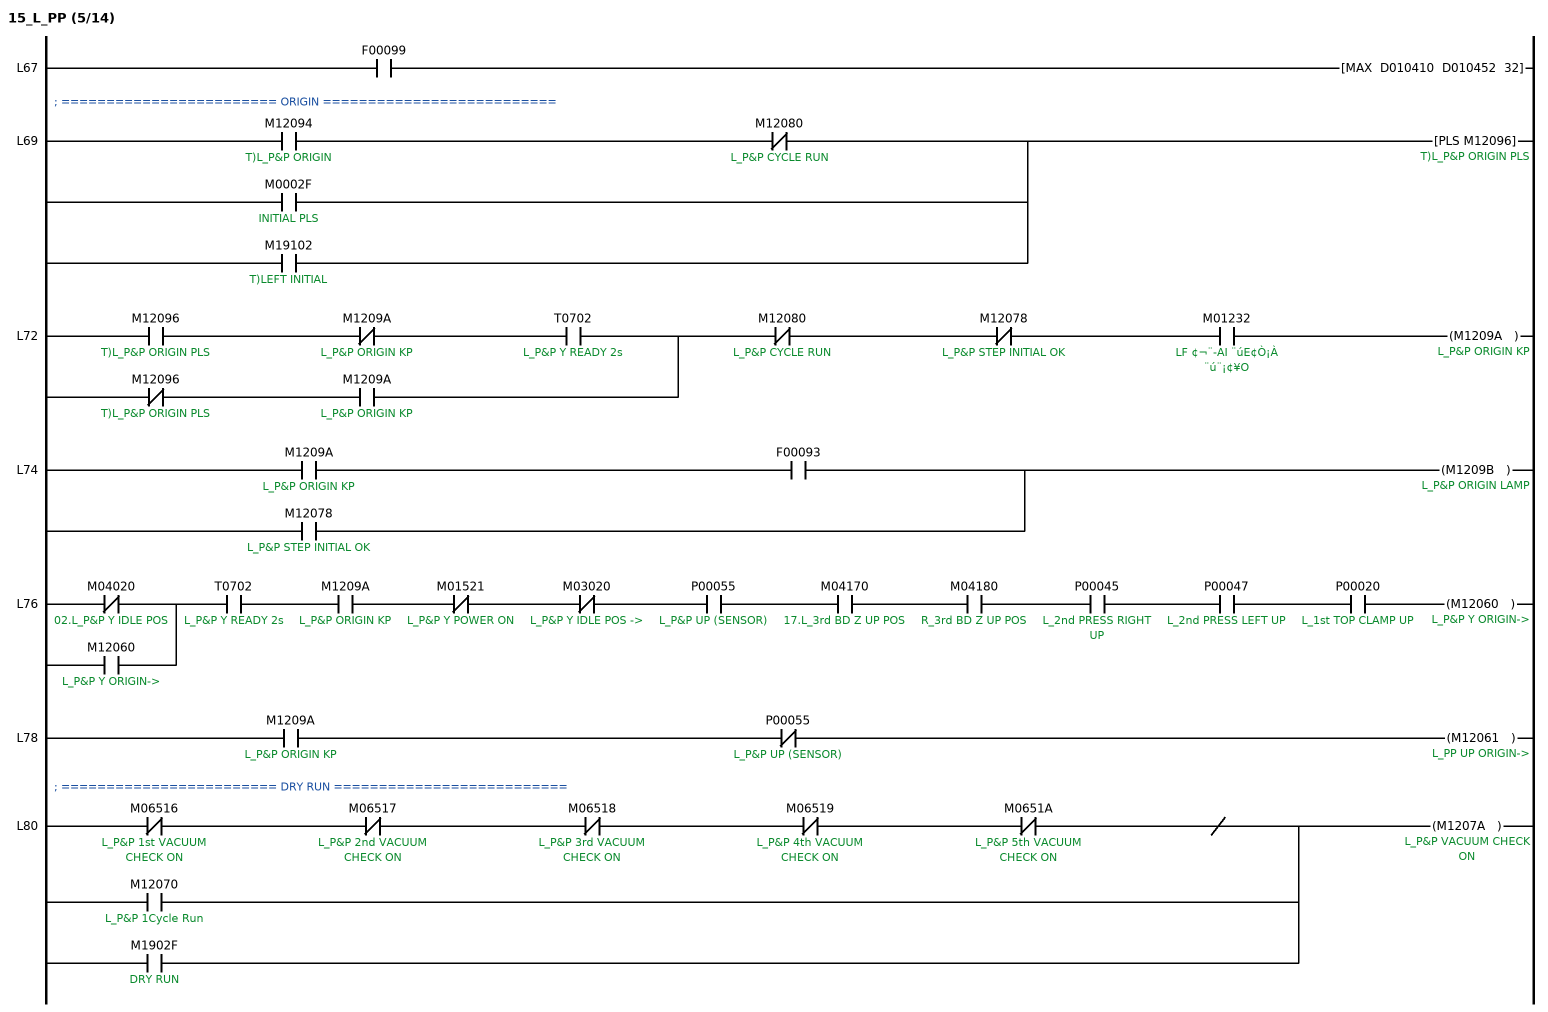
[picture p120: 15_L_PP rungs L67-L80]
; L67
LOAD      F00099
MAX       D010410 D010452 32
// ======================== ORIGIN ==========================
; L69
LOAD      M12094	// T)L_P&P ORIGIN
AND NOT   M12080	// L_P&P CYCLE RUN
OR        M0002F	// INITIAL PLS
OR        M19102	// T)LEFT INITIAL
OUTP      M12096	// T)L_P&P ORIGIN PLS
; L72
LOAD      M12096	// T)L_P&P ORIGIN PLS
AND NOT   M1209A	// L_P&P ORIGIN KP
AND       T0702	// L_P&P Y READY 2s
LOAD NOT  M12096	// T)L_P&P ORIGIN PLS
AND       M1209A	// L_P&P ORIGIN KP
OR LOAD
AND NOT   M12080	// L_P&P CYCLE RUN
AND NOT   M12078	// L_P&P STEP INITIAL OK
AND       M01232	// LF ¢¬¨­AI ¨úE¢Ò¡À ¨ú¨¡¢¥O
OUT       M1209A	// L_P&P ORIGIN KP
; L74
LOAD      M1209A	// L_P&P ORIGIN KP
AND       F00093
OR        M12078	// L_P&P STEP INITIAL OK
OUT       M1209B	// L_P&P ORIGIN LAMP
; L76
LOAD NOT  M04020	// 02.L_P&P Y IDLE POS
OR        M12060	// L_P&P Y ORIGIN->
AND       T0702	// L_P&P Y READY 2s
AND       M1209A	// L_P&P ORIGIN KP
AND NOT   M01521	// L_P&P Y POWER ON
AND NOT   M03020	// L_P&P Y IDLE POS ->
AND       P00055	// L_P&P UP (SENSOR)
AND       M04170	// 17.L_3rd BD Z UP POS
AND       M04180	// R_3rd BD Z UP POS
AND       P00045	// L_2nd PRESS RIGHT UP
AND       P00047	// L_2nd PRESS LEFT UP
AND       P00020	// L_1st TOP CLAMP UP
OUT       M12060	// L_P&P Y ORIGIN->
; L78
LOAD      M1209A	// L_P&P ORIGIN KP
AND NOT   P00055	// L_P&P UP (SENSOR)
OUT       M12061	// L_PP UP ORIGIN->
// ======================== DRY RUN ==========================
; L80
LOAD NOT  M06516	// L_P&P 1st VACUUM CHECK ON
AND NOT   M06517	// L_P&P 2nd VACUUM CHECK ON
AND NOT   M06518	// L_P&P 3rd VACUUM CHECK ON
AND NOT   M06519	// L_P&P 4th VACUUM CHECK ON
AND NOT   M0651A	// L_P&P 5th VACUUM CHECK ON
NOT
OR        M12070	// L_P&P 1Cycle Run
OR        M1902F	// DRY RUN
OUT       M1207A	// L_P&P VACUUM CHECK ON

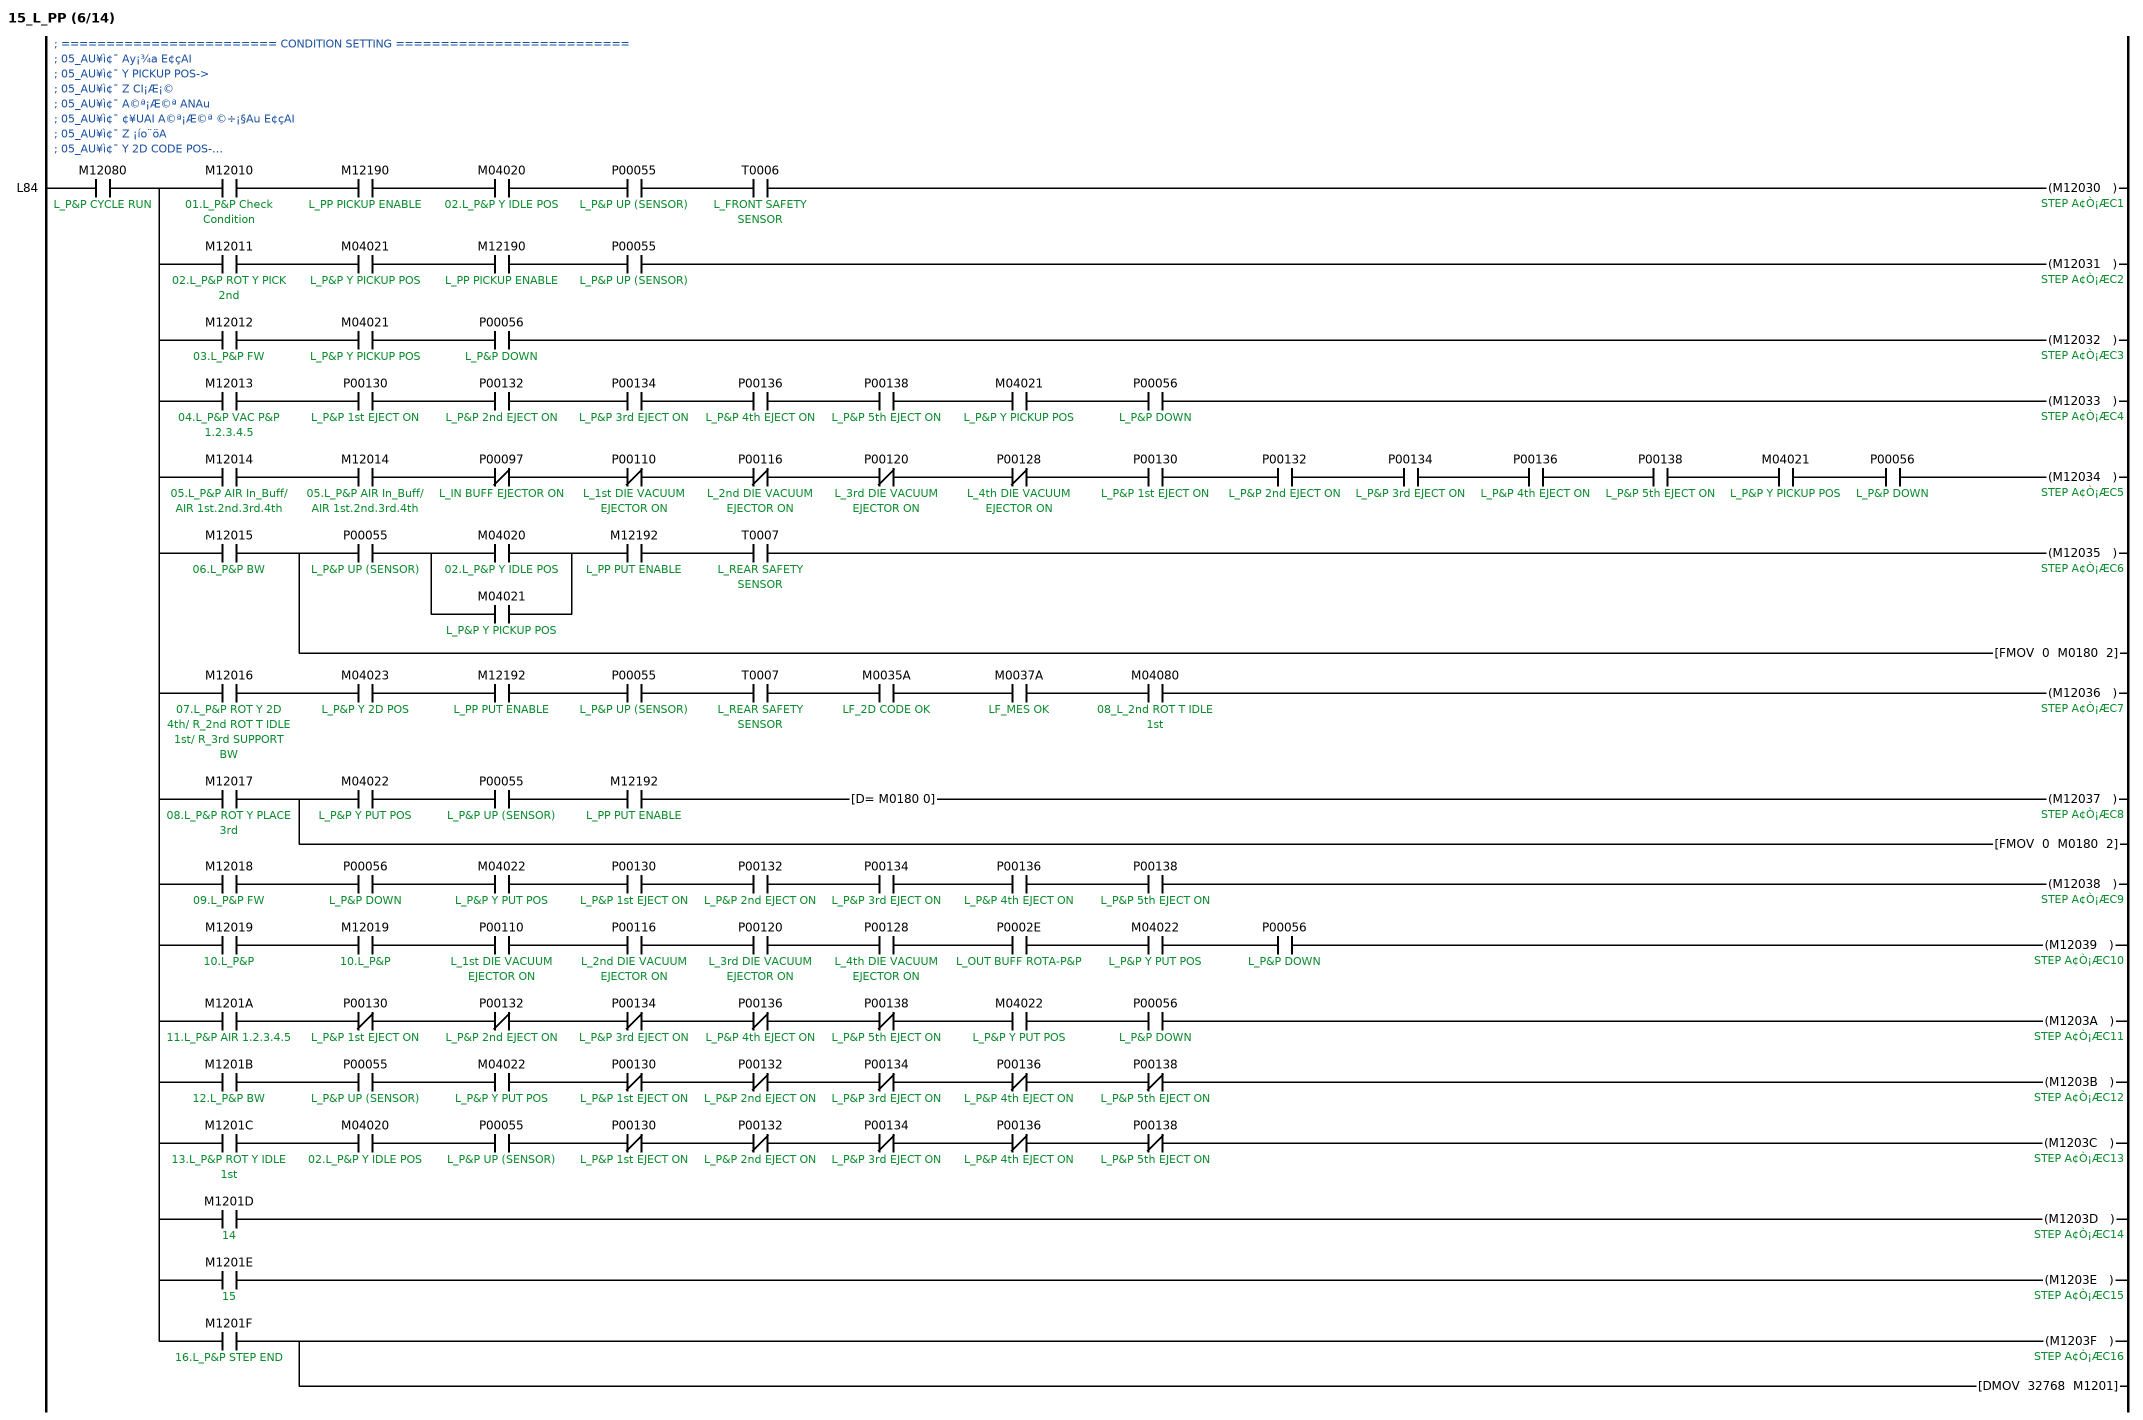
// ======================== CONDITION SETTING ==========================
; L84
LOAD      M12080	// L_P&P CYCLE RUN
MPUSH
AND       M12010	// 01.L_P&P Check Condition
AND       M12190	// L_PP PICKUP ENABLE
AND       M04020	// 02.L_P&P Y IDLE POS
AND       P00055	// L_P&P UP (SENSOR)
AND       T0006	// L_FRONT SAFETY SENSOR
OUT       M12030	// STEP A¢Ò¡ÆC1
MLOAD
AND       M12011	// 02.L_P&P ROT Y PICK 2nd
AND       M04021	// L_P&P Y PICKUP POS
AND       M12190	// L_PP PICKUP ENABLE
AND       P00055	// L_P&P UP (SENSOR)
OUT       M12031	// STEP A¢Ò¡ÆC2
MLOAD
AND       M12012	// 03.L_P&P FW
AND       M04021	// L_P&P Y PICKUP POS
AND       P00056	// L_P&P DOWN
OUT       M12032	// STEP A¢Ò¡ÆC3
MLOAD
AND       M12013	// 04.L_P&P VAC P&P 1.2.3.4.5
AND       P00130	// L_P&P 1st EJECT ON
AND       P00132	// L_P&P 2nd EJECT ON
AND       P00134	// L_P&P 3rd EJECT ON
AND       P00136	// L_P&P 4th EJECT ON
AND       P00138	// L_P&P 5th EJECT ON
AND       M04021	// L_P&P Y PICKUP POS
AND       P00056	// L_P&P DOWN
OUT       M12033	// STEP A¢Ò¡ÆC4
MLOAD
AND       M12014	// 05.L_P&P AIR In_Buff/ AIR 1st.2nd.3rd.4th
AND       M12014	// 05.L_P&P AIR In_Buff/ AIR 1st.2nd.3rd.4th
AND NOT   P00097	// L_IN BUFF EJECTOR ON
AND NOT   P00110	// L_1st DIE VACUUM EJECTOR ON
AND NOT   P00116	// L_2nd DIE VACUUM EJECTOR ON
AND NOT   P00120	// L_3rd DIE VACUUM EJECTOR ON
AND NOT   P00128	// L_4th DIE VACUUM EJECTOR ON
AND       P00130	// L_P&P 1st EJECT ON
AND       P00132	// L_P&P 2nd EJECT ON
AND       P00134	// L_P&P 3rd EJECT ON
AND       P00136	// L_P&P 4th EJECT ON
AND       P00138	// L_P&P 5th EJECT ON
AND       M04021	// L_P&P Y PICKUP POS
AND       P00056	// L_P&P DOWN
OUT       M12034	// STEP A¢Ò¡ÆC5
MLOAD
AND       M12015	// 06.L_P&P BW
MPUSH
AND       P00055	// L_P&P UP (SENSOR)
LOAD      M04020	// 02.L_P&P Y IDLE POS
OR        M04021	// L_P&P Y PICKUP POS
AND LOAD
AND       M12192	// L_PP PUT ENABLE
AND       T0007	// L_REAR SAFETY SENSOR
OUT       M12035	// STEP A¢Ò¡ÆC6
MPOP
FMOV      0 M0180 2
MLOAD
AND       M12016	// 07.L_P&P ROT Y 2D 4th/ R_2nd ROT T IDLE 1st/ R_3rd SUPPORT BW
AND       M04023	// L_P&P Y 2D POS
AND       M12192	// L_PP PUT ENABLE
AND       P00055	// L_P&P UP (SENSOR)
AND       T0007	// L_REAR SAFETY SENSOR
AND       M0035A	// LF_2D CODE OK
AND       M0037A	// LF_MES OK
AND       M04080	// 08_L_2nd ROT T IDLE 1st
OUT       M12036	// STEP A¢Ò¡ÆC7
MLOAD
AND       M12017	// 08.L_P&P ROT Y PLACE 3rd
MPUSH
AND       M04022	// L_P&P Y PUT POS
AND       P00055	// L_P&P UP (SENSOR)
AND       M12192	// L_PP PUT ENABLE
ANDD=     M0180 0
OUT       M12037	// STEP A¢Ò¡ÆC8
MPOP
FMOV      0 M0180 2
MLOAD
AND       M12018	// 09.L_P&P FW
AND       P00056	// L_P&P DOWN
AND       M04022	// L_P&P Y PUT POS
AND       P00130	// L_P&P 1st EJECT ON
AND       P00132	// L_P&P 2nd EJECT ON
AND       P00134	// L_P&P 3rd EJECT ON
AND       P00136	// L_P&P 4th EJECT ON
AND       P00138	// L_P&P 5th EJECT ON
OUT       M12038	// STEP A¢Ò¡ÆC9
MLOAD
AND       M12019	// 10.L_P&P
AND       M12019	// 10.L_P&P
AND       P00110	// L_1st DIE VACUUM EJECTOR ON
AND       P00116	// L_2nd DIE VACUUM EJECTOR ON
AND       P00120	// L_3rd DIE VACUUM EJECTOR ON
AND       P00128	// L_4th DIE VACUUM EJECTOR ON
AND       P0002E	// L_OUT BUFF ROTA-P&P
AND       M04022	// L_P&P Y PUT POS
AND       P00056	// L_P&P DOWN
OUT       M12039	// STEP A¢Ò¡ÆC10
MLOAD
AND       M1201A	// 11.L_P&P AIR 1.2.3.4.5
AND NOT   P00130	// L_P&P 1st EJECT ON
AND NOT   P00132	// L_P&P 2nd EJECT ON
AND NOT   P00134	// L_P&P 3rd EJECT ON
AND NOT   P00136	// L_P&P 4th EJECT ON
AND NOT   P00138	// L_P&P 5th EJECT ON
AND       M04022	// L_P&P Y PUT POS
AND       P00056	// L_P&P DOWN
OUT       M1203A	// STEP A¢Ò¡ÆC11
MLOAD
AND       M1201B	// 12.L_P&P BW
AND       P00055	// L_P&P UP (SENSOR)
AND       M04022	// L_P&P Y PUT POS
AND NOT   P00130	// L_P&P 1st EJECT ON
AND NOT   P00132	// L_P&P 2nd EJECT ON
AND NOT   P00134	// L_P&P 3rd EJECT ON
AND NOT   P00136	// L_P&P 4th EJECT ON
AND NOT   P00138	// L_P&P 5th EJECT ON
OUT       M1203B	// STEP A¢Ò¡ÆC12
MLOAD
AND       M1201C	// 13.L_P&P ROT Y IDLE 1st
AND       M04020	// 02.L_P&P Y IDLE POS
AND       P00055	// L_P&P UP (SENSOR)
AND NOT   P00130	// L_P&P 1st EJECT ON
AND NOT   P00132	// L_P&P 2nd EJECT ON
AND NOT   P00134	// L_P&P 3rd EJECT ON
AND NOT   P00136	// L_P&P 4th EJECT ON
AND NOT   P00138	// L_P&P 5th EJECT ON
OUT       M1203C	// STEP A¢Ò¡ÆC13
MLOAD
AND       M1201D	// 14
OUT       M1203D	// STEP A¢Ò¡ÆC14
MLOAD
AND       M1201E	// 15
OUT       M1203E	// STEP A¢Ò¡ÆC15
MPOP
AND       M1201F	// 16.L_P&P STEP END
OUT       M1203F	// STEP A¢Ò¡ÆC16
DMOV      32768 M1201
// output comment: 05_AU¥ì¢¯ Ay¡¾a E¢çAI
// output comment: 05_AU¥ì¢¯ Y PICKUP POS->
// output comment: 05_AU¥ì¢¯ Z CI¡Æ¡©
// output comment: 05_AU¥ì¢¯ A©ª¡Æ©ª ANAu
// output comment: 05_AU¥ì¢¯ ¢¥UAI A©ª¡Æ©ª ©÷¡§Au E¢çAI
// output comment: 05_AU¥ì¢¯ Z ¡ío¨öA
// output comment: 05_AU¥ì¢¯ Y 2D CODE POS->
// output comment: 05_AU¥ì¢¯ Y PUT POS->
// output comment: 05_AU¥ì¢¯ Z CI¡Æ¡©
// output comment: 05_AU¥ì¢¯ A©ª¡Æ©ª ANAu E¢çAI
// output comment: 05_AU¥ì¢¯ A©ª¡Æ©ª ©÷¡§Au
// output comment: 05_AU¥ì¢¯ Z ¡ío¨öA
// output comment: 05_AU¥ì¢¯ Y IDLE POS->

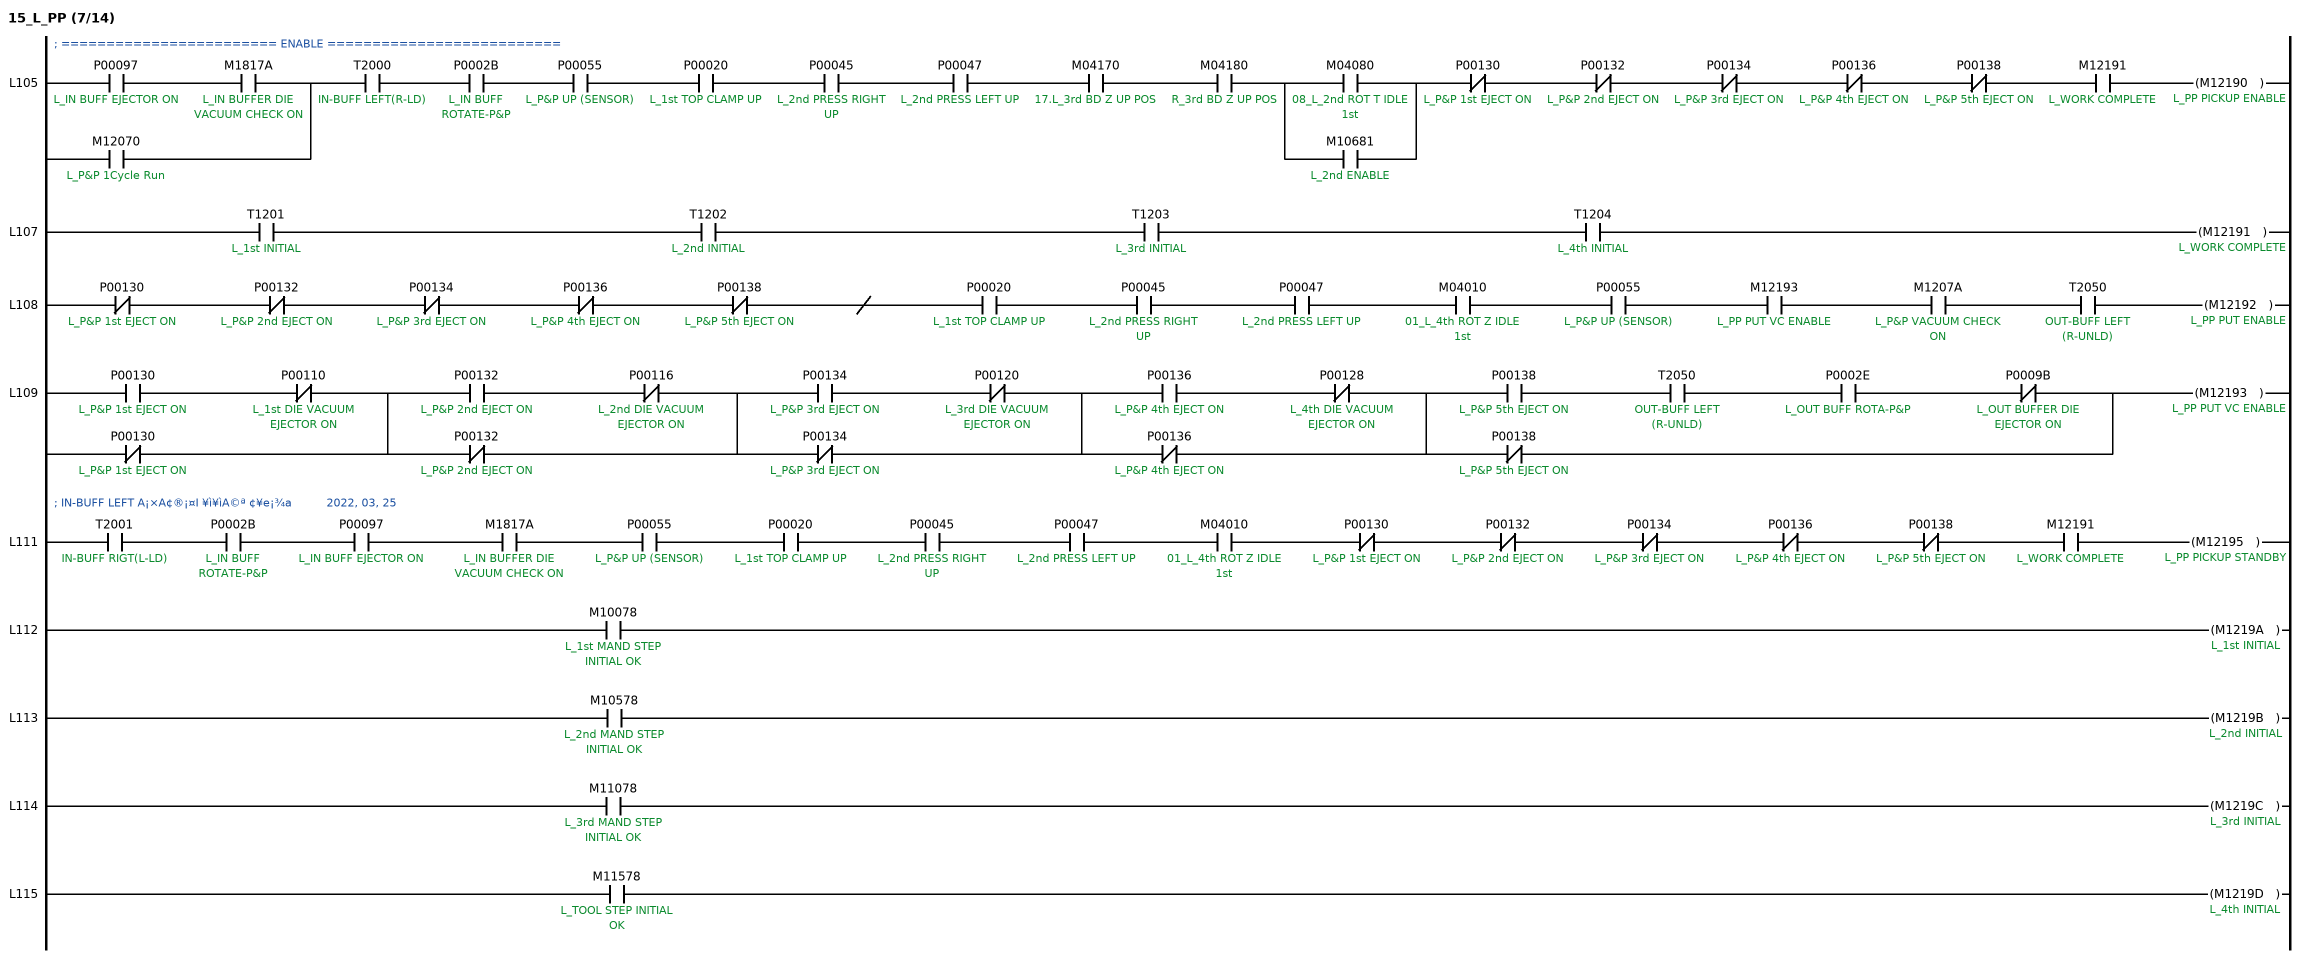
// ======================== ENABLE ==========================
; L105
LOAD      P00097	// L_IN BUFF EJECTOR ON
AND       M1817A	// L_IN BUFFER DIE VACUUM CHECK ON
OR        M12070	// L_P&P 1Cycle Run
AND       T2000	// IN-BUFF LEFT(R-LD)
AND       P0002B	// L_IN BUFF ROTATE-P&P
AND       P00055	// L_P&P UP (SENSOR)
AND       P00020	// L_1st TOP CLAMP UP
AND       P00045	// L_2nd PRESS RIGHT UP
AND       P00047	// L_2nd PRESS LEFT UP
AND       M04170	// 17.L_3rd BD Z UP POS
AND       M04180	// R_3rd BD Z UP POS
LOAD      M04080	// 08_L_2nd ROT T IDLE 1st
OR        M10681	// L_2nd ENABLE
AND LOAD
AND NOT   P00130	// L_P&P 1st EJECT ON
AND NOT   P00132	// L_P&P 2nd EJECT ON
AND NOT   P00134	// L_P&P 3rd EJECT ON
AND NOT   P00136	// L_P&P 4th EJECT ON
AND NOT   P00138	// L_P&P 5th EJECT ON
AND       M12191	// L_WORK COMPLETE
OUT       M12190	// L_PP PICKUP ENABLE
; L107
LOAD      T1201	// L_1st INITIAL
AND       T1202	// L_2nd INITIAL
AND       T1203	// L_3rd INITIAL
AND       T1204	// L_4th INITIAL
OUT       M12191	// L_WORK COMPLETE
; L108
LOAD NOT  P00130	// L_P&P 1st EJECT ON
AND NOT   P00132	// L_P&P 2nd EJECT ON
AND NOT   P00134	// L_P&P 3rd EJECT ON
AND NOT   P00136	// L_P&P 4th EJECT ON
AND NOT   P00138	// L_P&P 5th EJECT ON
NOT
AND       P00020	// L_1st TOP CLAMP UP
AND       P00045	// L_2nd PRESS RIGHT UP
AND       P00047	// L_2nd PRESS LEFT UP
AND       M04010	// 01_L_4th ROT Z IDLE 1st
AND       P00055	// L_P&P UP (SENSOR)
AND       M12193	// L_PP PUT VC ENABLE
AND       M1207A	// L_P&P VACUUM CHECK ON
AND       T2050	// OUT-BUFF LEFT (R-UNLD)
OUT       M12192	// L_PP PUT ENABLE
; L109
LOAD      P00130	// L_P&P 1st EJECT ON
AND NOT   P00110	// L_1st DIE VACUUM EJECTOR ON
OR NOT    P00130	// L_P&P 1st EJECT ON
LOAD      P00132	// L_P&P 2nd EJECT ON
AND NOT   P00116	// L_2nd DIE VACUUM EJECTOR ON
OR NOT    P00132	// L_P&P 2nd EJECT ON
AND LOAD
LOAD      P00134	// L_P&P 3rd EJECT ON
AND NOT   P00120	// L_3rd DIE VACUUM EJECTOR ON
OR NOT    P00134	// L_P&P 3rd EJECT ON
AND LOAD
LOAD      P00136	// L_P&P 4th EJECT ON
AND NOT   P00128	// L_4th DIE VACUUM EJECTOR ON
OR NOT    P00136	// L_P&P 4th EJECT ON
AND LOAD
LOAD      P00138	// L_P&P 5th EJECT ON
AND       T2050	// OUT-BUFF LEFT (R-UNLD)
AND       P0002E	// L_OUT BUFF ROTA-P&P
AND NOT   P0009B	// L_OUT BUFFER DIE EJECTOR ON
OR NOT    P00138	// L_P&P 5th EJECT ON
AND LOAD
OUT       M12193	// L_PP PUT VC ENABLE
; L111
LOAD      T2001	// IN-BUFF RIGT(L-LD)
AND       P0002B	// L_IN BUFF ROTATE-P&P
AND       P00097	// L_IN BUFF EJECTOR ON
AND       M1817A	// L_IN BUFFER DIE VACUUM CHECK ON
AND       P00055	// L_P&P UP (SENSOR)
AND       P00020	// L_1st TOP CLAMP UP
AND       P00045	// L_2nd PRESS RIGHT UP
AND       P00047	// L_2nd PRESS LEFT UP
AND       M04010	// 01_L_4th ROT Z IDLE 1st
AND NOT   P00130	// L_P&P 1st EJECT ON
AND NOT   P00132	// L_P&P 2nd EJECT ON
AND NOT   P00134	// L_P&P 3rd EJECT ON
AND NOT   P00136	// L_P&P 4th EJECT ON
AND NOT   P00138	// L_P&P 5th EJECT ON
AND       M12191	// L_WORK COMPLETE
OUT       M12195	// L_PP PICKUP STANDBY
// output comment: IN-BUFF LEFT A¡×A¢®¡¤I ¥ì¥ìA©ª ¢¥e¡¾a          2022, 03, 25
; L112
LOAD      M10078	// L_1st MAND STEP INITIAL OK
OUT       M1219A	// L_1st INITIAL
; L113
LOAD      M10578	// L_2nd MAND STEP INITIAL OK
OUT       M1219B	// L_2nd INITIAL
; L114
LOAD      M11078	// L_3rd MAND STEP INITIAL OK
OUT       M1219C	// L_3rd INITIAL
; L115
LOAD      M11578	// L_TOOL STEP INITIAL OK
OUT       M1219D	// L_4th INITIAL

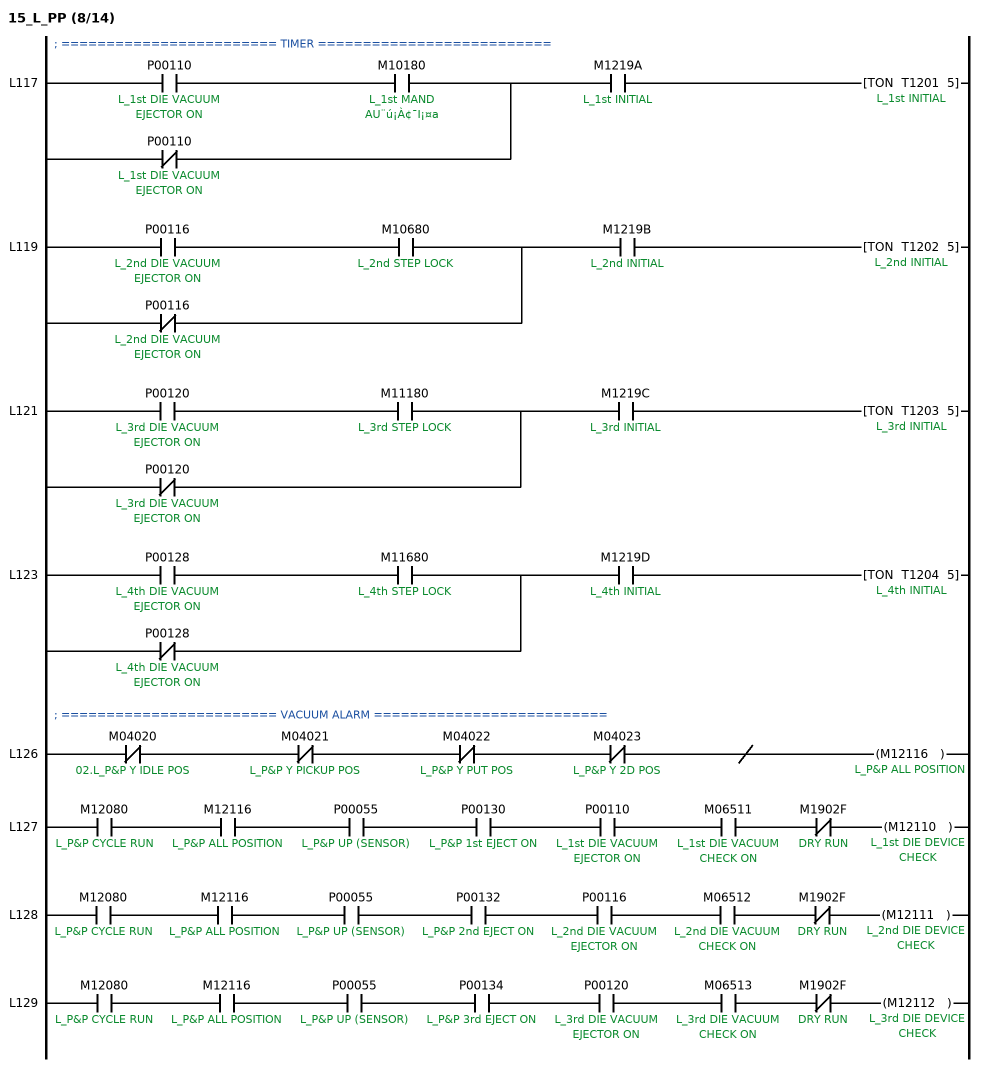
// ======================== TIMER ==========================
; L117
LOAD      P00110	// L_1st DIE VACUUM EJECTOR ON
AND       M10180	// L_1st MAND AU¨ú¡À¢¯I¡¤a
OR NOT    P00110	// L_1st DIE VACUUM EJECTOR ON
AND       M1219A	// L_1st INITIAL
TON       T1201 5	// L_1st INITIAL
; L119
LOAD      P00116	// L_2nd DIE VACUUM EJECTOR ON
AND       M10680	// L_2nd STEP LOCK
OR NOT    P00116	// L_2nd DIE VACUUM EJECTOR ON
AND       M1219B	// L_2nd INITIAL
TON       T1202 5	// L_2nd INITIAL
; L121
LOAD      P00120	// L_3rd DIE VACUUM EJECTOR ON
AND       M11180	// L_3rd STEP LOCK
OR NOT    P00120	// L_3rd DIE VACUUM EJECTOR ON
AND       M1219C	// L_3rd INITIAL
TON       T1203 5	// L_3rd INITIAL
; L123
LOAD      P00128	// L_4th DIE VACUUM EJECTOR ON
AND       M11680	// L_4th STEP LOCK
OR NOT    P00128	// L_4th DIE VACUUM EJECTOR ON
AND       M1219D	// L_4th INITIAL
TON       T1204 5	// L_4th INITIAL
// ======================== VACUUM ALARM ==========================
; L126
LOAD NOT  M04020	// 02.L_P&P Y IDLE POS
AND NOT   M04021	// L_P&P Y PICKUP POS
AND NOT   M04022	// L_P&P Y PUT POS
AND NOT   M04023	// L_P&P Y 2D POS
NOT
OUT       M12116	// L_P&P ALL POSITION
; L127
LOAD      M12080	// L_P&P CYCLE RUN
AND       M12116	// L_P&P ALL POSITION
AND       P00055	// L_P&P UP (SENSOR)
AND       P00130	// L_P&P 1st EJECT ON
AND       P00110	// L_1st DIE VACUUM EJECTOR ON
AND       M06511	// L_1st DIE VACUUM CHECK ON
AND NOT   M1902F	// DRY RUN
OUT       M12110	// L_1st DIE DEVICE CHECK
; L128
LOAD      M12080	// L_P&P CYCLE RUN
AND       M12116	// L_P&P ALL POSITION
AND       P00055	// L_P&P UP (SENSOR)
AND       P00132	// L_P&P 2nd EJECT ON
AND       P00116	// L_2nd DIE VACUUM EJECTOR ON
AND       M06512	// L_2nd DIE VACUUM CHECK ON
AND NOT   M1902F	// DRY RUN
OUT       M12111	// L_2nd DIE DEVICE CHECK
; L129
LOAD      M12080	// L_P&P CYCLE RUN
AND       M12116	// L_P&P ALL POSITION
AND       P00055	// L_P&P UP (SENSOR)
AND       P00134	// L_P&P 3rd EJECT ON
AND       P00120	// L_3rd DIE VACUUM EJECTOR ON
AND       M06513	// L_3rd DIE VACUUM CHECK ON
AND NOT   M1902F	// DRY RUN
OUT       M12112	// L_3rd DIE DEVICE CHECK

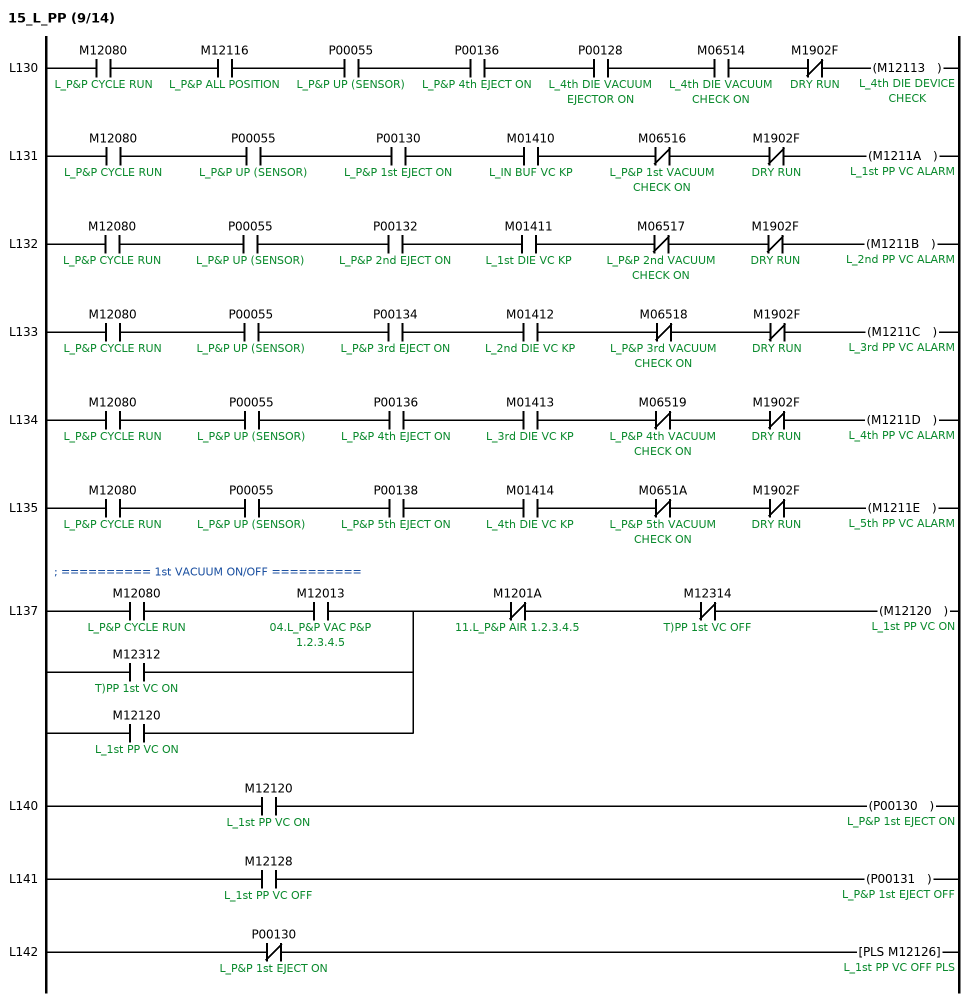
; L130
LOAD      M12080	// L_P&P CYCLE RUN
AND       M12116	// L_P&P ALL POSITION
AND       P00055	// L_P&P UP (SENSOR)
AND       P00136	// L_P&P 4th EJECT ON
AND       P00128	// L_4th DIE VACUUM EJECTOR ON
AND       M06514	// L_4th DIE VACUUM CHECK ON
AND NOT   M1902F	// DRY RUN
OUT       M12113	// L_4th DIE DEVICE CHECK
; L131
LOAD      M12080	// L_P&P CYCLE RUN
AND       P00055	// L_P&P UP (SENSOR)
AND       P00130	// L_P&P 1st EJECT ON
AND       M01410	// L_IN BUF VC KP
AND NOT   M06516	// L_P&P 1st VACUUM CHECK ON
AND NOT   M1902F	// DRY RUN
OUT       M1211A	// L_1st PP VC ALARM
; L132
LOAD      M12080	// L_P&P CYCLE RUN
AND       P00055	// L_P&P UP (SENSOR)
AND       P00132	// L_P&P 2nd EJECT ON
AND       M01411	// L_1st DIE VC KP
AND NOT   M06517	// L_P&P 2nd VACUUM CHECK ON
AND NOT   M1902F	// DRY RUN
OUT       M1211B	// L_2nd PP VC ALARM
; L133
LOAD      M12080	// L_P&P CYCLE RUN
AND       P00055	// L_P&P UP (SENSOR)
AND       P00134	// L_P&P 3rd EJECT ON
AND       M01412	// L_2nd DIE VC KP
AND NOT   M06518	// L_P&P 3rd VACUUM CHECK ON
AND NOT   M1902F	// DRY RUN
OUT       M1211C	// L_3rd PP VC ALARM
; L134
LOAD      M12080	// L_P&P CYCLE RUN
AND       P00055	// L_P&P UP (SENSOR)
AND       P00136	// L_P&P 4th EJECT ON
AND       M01413	// L_3rd DIE VC KP
AND NOT   M06519	// L_P&P 4th VACUUM CHECK ON
AND NOT   M1902F	// DRY RUN
OUT       M1211D	// L_4th PP VC ALARM
; L135
LOAD      M12080	// L_P&P CYCLE RUN
AND       P00055	// L_P&P UP (SENSOR)
AND       P00138	// L_P&P 5th EJECT ON
AND       M01414	// L_4th DIE VC KP
AND NOT   M0651A	// L_P&P 5th VACUUM CHECK ON
AND NOT   M1902F	// DRY RUN
OUT       M1211E	// L_5th PP VC ALARM
// ========== 1st VACUUM ON/OFF ==========
; L137
LOAD      M12080	// L_P&P CYCLE RUN
AND       M12013	// 04.L_P&P VAC P&P 1.2.3.4.5
OR        M12312	// T)PP 1st VC ON
OR        M12120	// L_1st PP VC ON
AND NOT   M1201A	// 11.L_P&P AIR 1.2.3.4.5
AND NOT   M12314	// T)PP 1st VC OFF
OUT       M12120	// L_1st PP VC ON
; L140
LOAD      M12120	// L_1st PP VC ON
OUT       P00130	// L_P&P 1st EJECT ON
; L141
LOAD      M12128	// L_1st PP VC OFF
OUT       P00131	// L_P&P 1st EJECT OFF
; L142
LOAD NOT  P00130	// L_P&P 1st EJECT ON
OUTP      M12126	// L_1st PP VC OFF PLS

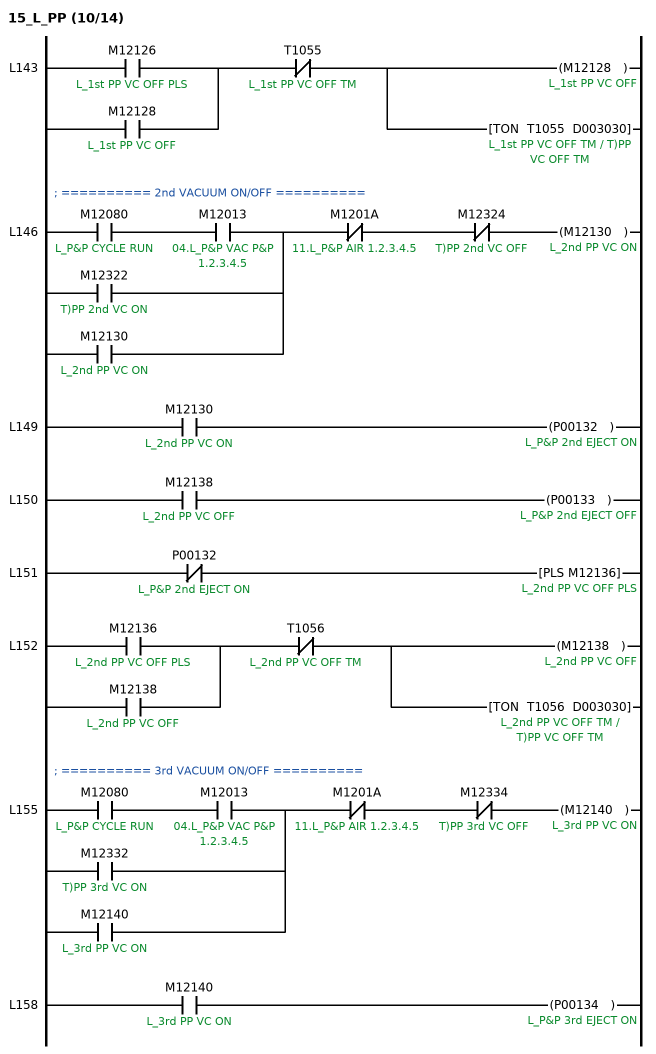
; L143
LOAD      M12126	// L_1st PP VC OFF PLS
OR        M12128	// L_1st PP VC OFF
AND NOT   T1055	// L_1st PP VC OFF TM
OUT       M12128	// L_1st PP VC OFF
TON       T1055 D003030	// L_1st PP VC OFF TM / T)PP VC OFF TM
// ========== 2nd VACUUM ON/OFF ==========
; L146
LOAD      M12080	// L_P&P CYCLE RUN
AND       M12013	// 04.L_P&P VAC P&P 1.2.3.4.5
OR        M12322	// T)PP 2nd VC ON
OR        M12130	// L_2nd PP VC ON
AND NOT   M1201A	// 11.L_P&P AIR 1.2.3.4.5
AND NOT   M12324	// T)PP 2nd VC OFF
OUT       M12130	// L_2nd PP VC ON
; L149
LOAD      M12130	// L_2nd PP VC ON
OUT       P00132	// L_P&P 2nd EJECT ON
; L150
LOAD      M12138	// L_2nd PP VC OFF
OUT       P00133	// L_P&P 2nd EJECT OFF
; L151
LOAD NOT  P00132	// L_P&P 2nd EJECT ON
OUTP      M12136	// L_2nd PP VC OFF PLS
; L152
LOAD      M12136	// L_2nd PP VC OFF PLS
OR        M12138	// L_2nd PP VC OFF
AND NOT   T1056	// L_2nd PP VC OFF TM
OUT       M12138	// L_2nd PP VC OFF
TON       T1056 D003030	// L_2nd PP VC OFF TM / T)PP VC OFF TM
// ========== 3rd VACUUM ON/OFF ==========
; L155
LOAD      M12080	// L_P&P CYCLE RUN
AND       M12013	// 04.L_P&P VAC P&P 1.2.3.4.5
OR        M12332	// T)PP 3rd VC ON
OR        M12140	// L_3rd PP VC ON
AND NOT   M1201A	// 11.L_P&P AIR 1.2.3.4.5
AND NOT   M12334	// T)PP 3rd VC OFF
OUT       M12140	// L_3rd PP VC ON
; L158
LOAD      M12140	// L_3rd PP VC ON
OUT       P00134	// L_P&P 3rd EJECT ON

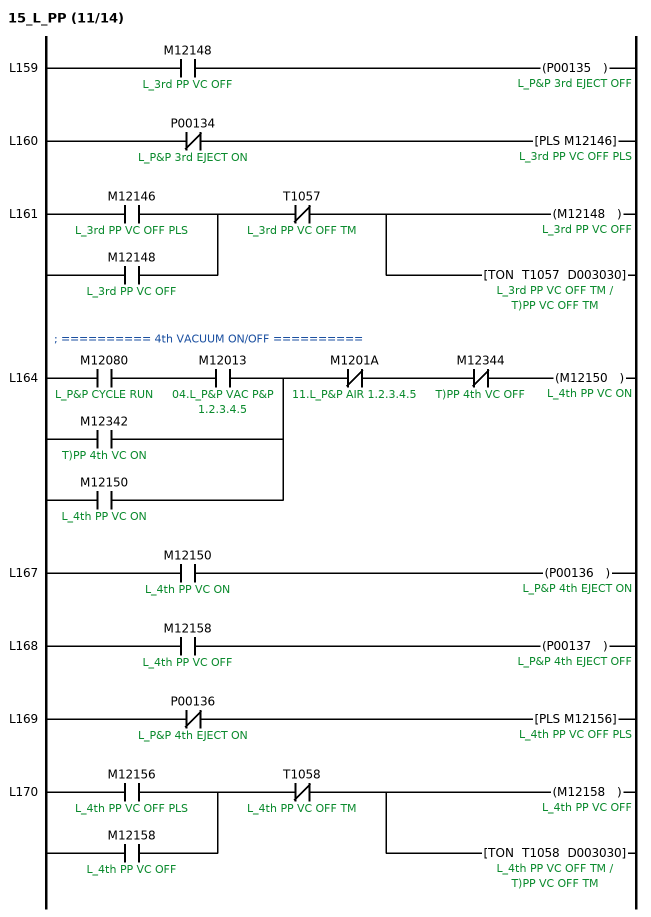
; L159
LOAD      M12148	// L_3rd PP VC OFF
OUT       P00135	// L_P&P 3rd EJECT OFF
; L160
LOAD NOT  P00134	// L_P&P 3rd EJECT ON
OUTP      M12146	// L_3rd PP VC OFF PLS
; L161
LOAD      M12146	// L_3rd PP VC OFF PLS
OR        M12148	// L_3rd PP VC OFF
AND NOT   T1057	// L_3rd PP VC OFF TM
OUT       M12148	// L_3rd PP VC OFF
TON       T1057 D003030	// L_3rd PP VC OFF TM / T)PP VC OFF TM
// ========== 4th VACUUM ON/OFF ==========
; L164
LOAD      M12080	// L_P&P CYCLE RUN
AND       M12013	// 04.L_P&P VAC P&P 1.2.3.4.5
OR        M12342	// T)PP 4th VC ON
OR        M12150	// L_4th PP VC ON
AND NOT   M1201A	// 11.L_P&P AIR 1.2.3.4.5
AND NOT   M12344	// T)PP 4th VC OFF
OUT       M12150	// L_4th PP VC ON
; L167
LOAD      M12150	// L_4th PP VC ON
OUT       P00136	// L_P&P 4th EJECT ON
; L168
LOAD      M12158	// L_4th PP VC OFF
OUT       P00137	// L_P&P 4th EJECT OFF
; L169
LOAD NOT  P00136	// L_P&P 4th EJECT ON
OUTP      M12156	// L_4th PP VC OFF PLS
; L170
LOAD      M12156	// L_4th PP VC OFF PLS
OR        M12158	// L_4th PP VC OFF
AND NOT   T1058	// L_4th PP VC OFF TM
OUT       M12158	// L_4th PP VC OFF
TON       T1058 D003030	// L_4th PP VC OFF TM / T)PP VC OFF TM

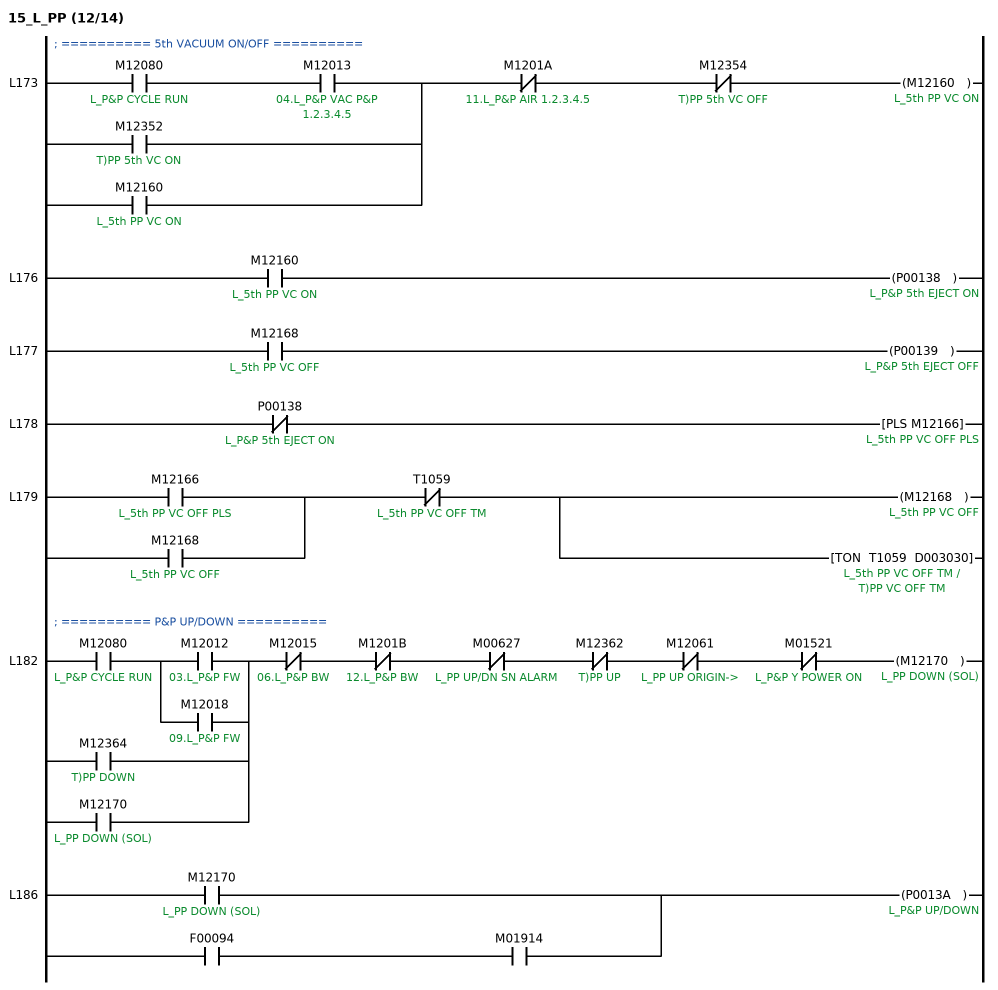
// ========== 5th VACUUM ON/OFF ==========
; L173
LOAD      M12080	// L_P&P CYCLE RUN
AND       M12013	// 04.L_P&P VAC P&P 1.2.3.4.5
OR        M12352	// T)PP 5th VC ON
OR        M12160	// L_5th PP VC ON
AND NOT   M1201A	// 11.L_P&P AIR 1.2.3.4.5
AND NOT   M12354	// T)PP 5th VC OFF
OUT       M12160	// L_5th PP VC ON
; L176
LOAD      M12160	// L_5th PP VC ON
OUT       P00138	// L_P&P 5th EJECT ON
; L177
LOAD      M12168	// L_5th PP VC OFF
OUT       P00139	// L_P&P 5th EJECT OFF
; L178
LOAD NOT  P00138	// L_P&P 5th EJECT ON
OUTP      M12166	// L_5th PP VC OFF PLS
; L179
LOAD      M12166	// L_5th PP VC OFF PLS
OR        M12168	// L_5th PP VC OFF
AND NOT   T1059	// L_5th PP VC OFF TM
OUT       M12168	// L_5th PP VC OFF
TON       T1059 D003030	// L_5th PP VC OFF TM / T)PP VC OFF TM
// ========== P&P UP/DOWN ==========
; L182
LOAD      M12080	// L_P&P CYCLE RUN
LOAD      M12012	// 03.L_P&P FW
OR        M12018	// 09.L_P&P FW
AND LOAD
OR        M12364	// T)PP DOWN
OR        M12170	// L_PP DOWN (SOL)
AND NOT   M12015	// 06.L_P&P BW
AND NOT   M1201B	// 12.L_P&P BW
AND NOT   M00627	// L_PP UP/DN SN ALARM
AND NOT   M12362	// T)PP UP
AND NOT   M12061	// L_PP UP ORIGIN->
AND NOT   M01521	// L_P&P Y POWER ON
OUT       M12170	// L_PP DOWN (SOL)
; L186
LOAD      M12170	// L_PP DOWN (SOL)
LOAD      F00094
AND       M01914
OR LOAD
OUT       P0013A	// L_P&P UP/DOWN

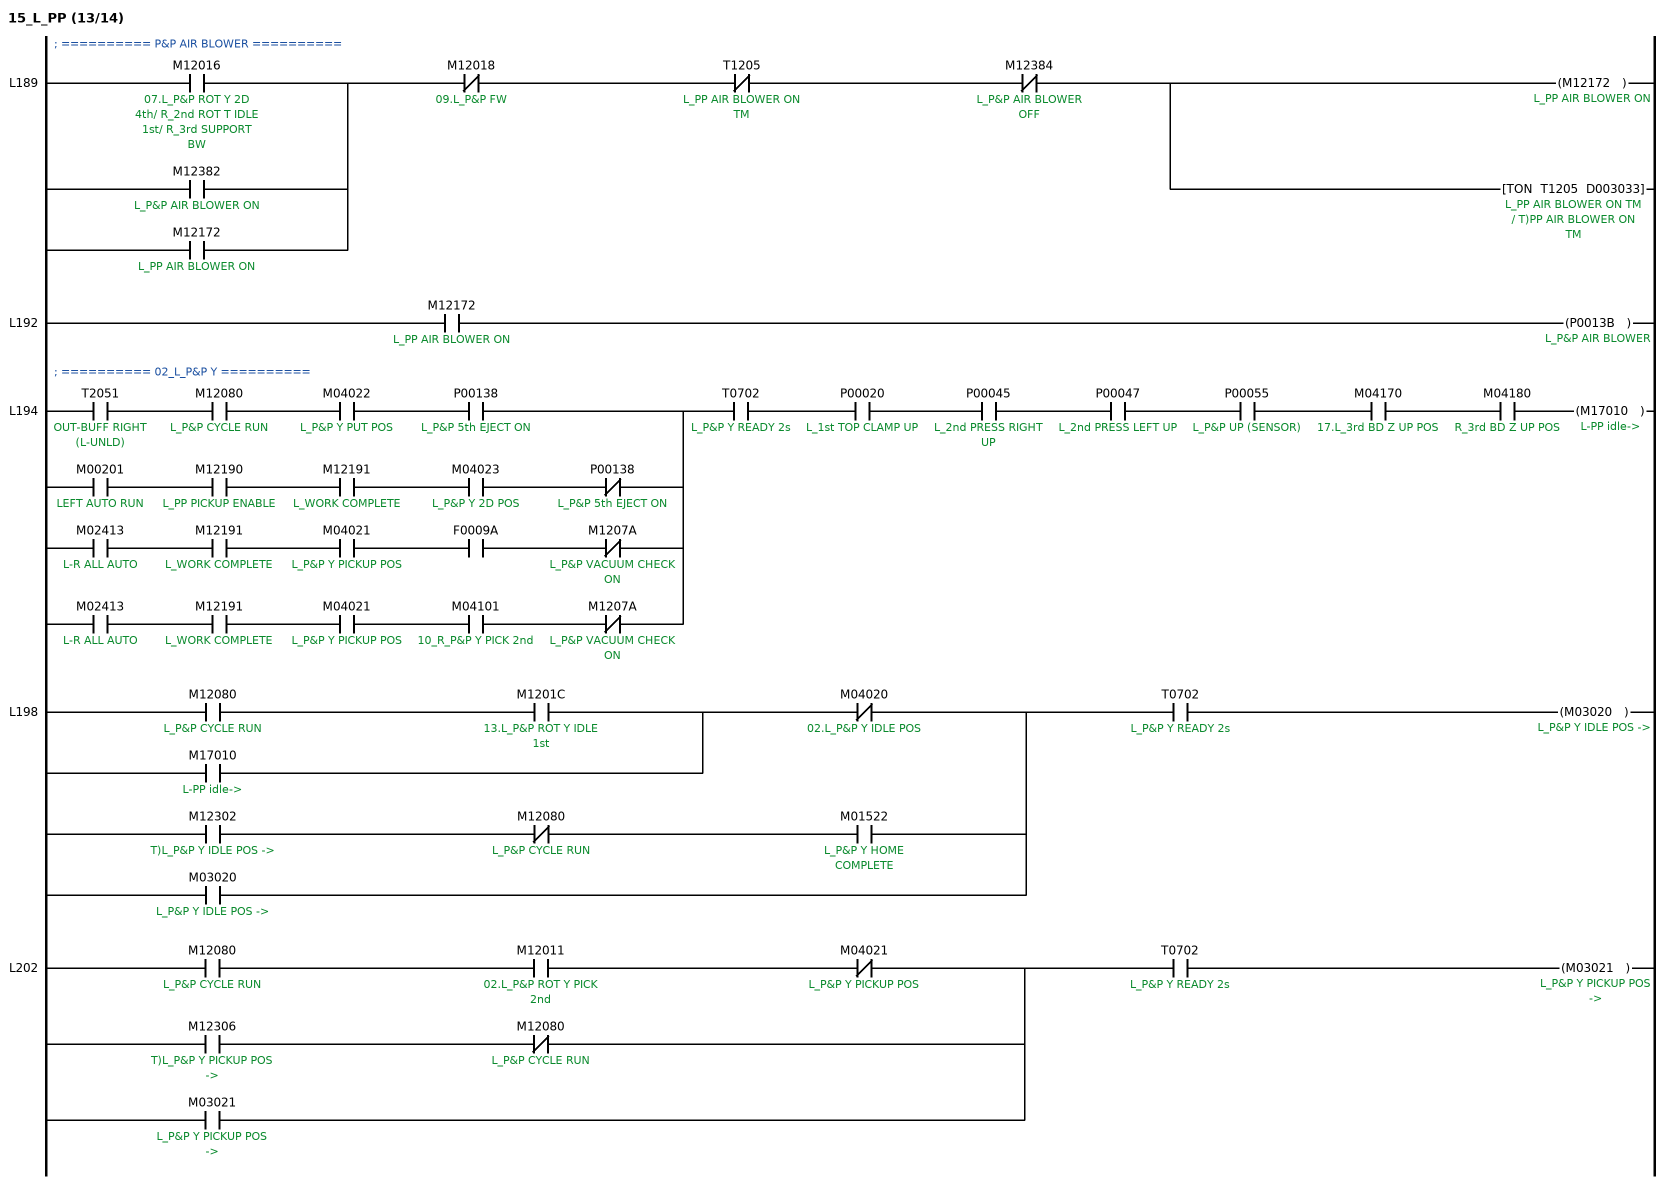
// ========== P&P AIR BLOWER ==========
; L189
LOAD      M12016	// 07.L_P&P ROT Y 2D 4th/ R_2nd ROT T IDLE 1st/ R_3rd SUPPORT BW
OR        M12382	// L_P&P AIR BLOWER ON
OR        M12172	// L_PP AIR BLOWER ON
AND NOT   M12018	// 09.L_P&P FW
AND NOT   T1205	// L_PP AIR BLOWER ON TM
AND NOT   M12384	// L_P&P AIR BLOWER OFF
OUT       M12172	// L_PP AIR BLOWER ON
TON       T1205 D003033	// L_PP AIR BLOWER ON TM / T)PP AIR BLOWER ON TM
; L192
LOAD      M12172	// L_PP AIR BLOWER ON
OUT       P0013B	// L_P&P AIR BLOWER
// ========== 02_L_P&P Y ==========
; L194
LOAD      T2051	// OUT-BUFF RIGHT (L-UNLD)
AND       M12080	// L_P&P CYCLE RUN
AND       M04022	// L_P&P Y PUT POS
AND       P00138	// L_P&P 5th EJECT ON
LOAD      M00201	// LEFT AUTO RUN
AND       M12190	// L_PP PICKUP ENABLE
AND       M12191	// L_WORK COMPLETE
AND       M04023	// L_P&P Y 2D POS
AND NOT   P00138	// L_P&P 5th EJECT ON
OR LOAD
LOAD      M02413	// L-R ALL AUTO
AND       M12191	// L_WORK COMPLETE
AND       M04021	// L_P&P Y PICKUP POS
AND       F0009A
AND NOT   M1207A	// L_P&P VACUUM CHECK ON
OR LOAD
LOAD      M02413	// L-R ALL AUTO
AND       M12191	// L_WORK COMPLETE
AND       M04021	// L_P&P Y PICKUP POS
AND       M04101	// 10_R_P&P Y PICK 2nd
AND NOT   M1207A	// L_P&P VACUUM CHECK ON
OR LOAD
AND       T0702	// L_P&P Y READY 2s
AND       P00020	// L_1st TOP CLAMP UP
AND       P00045	// L_2nd PRESS RIGHT UP
AND       P00047	// L_2nd PRESS LEFT UP
AND       P00055	// L_P&P UP (SENSOR)
AND       M04170	// 17.L_3rd BD Z UP POS
AND       M04180	// R_3rd BD Z UP POS
OUT       M17010	// L-PP idle->
; L198
LOAD      M12080	// L_P&P CYCLE RUN
AND       M1201C	// 13.L_P&P ROT Y IDLE 1st
OR        M17010	// L-PP idle->
AND NOT   M04020	// 02.L_P&P Y IDLE POS
LOAD      M12302	// T)L_P&P Y IDLE POS ->
AND NOT   M12080	// L_P&P CYCLE RUN
AND       M01522	// L_P&P Y HOME COMPLETE
OR LOAD
OR        M03020	// L_P&P Y IDLE POS ->
AND       T0702	// L_P&P Y READY 2s
OUT       M03020	// L_P&P Y IDLE POS ->
; L202
LOAD      M12080	// L_P&P CYCLE RUN
AND       M12011	// 02.L_P&P ROT Y PICK 2nd
AND NOT   M04021	// L_P&P Y PICKUP POS
LOAD      M12306	// T)L_P&P Y PICKUP POS ->
AND NOT   M12080	// L_P&P CYCLE RUN
OR LOAD
OR        M03021	// L_P&P Y PICKUP POS ->
AND       T0702	// L_P&P Y READY 2s
OUT       M03021	// L_P&P Y PICKUP POS ->

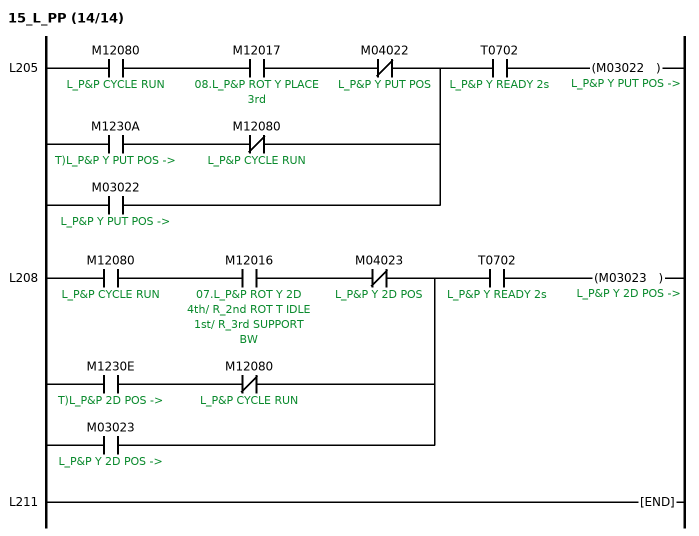
; L205
LOAD      M12080	// L_P&P CYCLE RUN
AND       M12017	// 08.L_P&P ROT Y PLACE 3rd
AND NOT   M04022	// L_P&P Y PUT POS
LOAD      M1230A	// T)L_P&P Y PUT POS ->
AND NOT   M12080	// L_P&P CYCLE RUN
OR LOAD
OR        M03022	// L_P&P Y PUT POS ->
AND       T0702	// L_P&P Y READY 2s
OUT       M03022	// L_P&P Y PUT POS ->
; L208
LOAD      M12080	// L_P&P CYCLE RUN
AND       M12016	// 07.L_P&P ROT Y 2D 4th/ R_2nd ROT T IDLE 1st/ R_3rd SUPPORT BW
AND NOT   M04023	// L_P&P Y 2D POS
LOAD      M1230E	// T)L_P&P 2D POS ->
AND NOT   M12080	// L_P&P CYCLE RUN
OR LOAD
OR        M03023	// L_P&P Y 2D POS ->
AND       T0702	// L_P&P Y READY 2s
OUT       M03023	// L_P&P Y 2D POS ->
; L211
END

PROGRAM 16_R_1st_MAND (task: ¨ö¨¬A¥ì CA¡¤I¡¾¡¿¡¤¡Í)

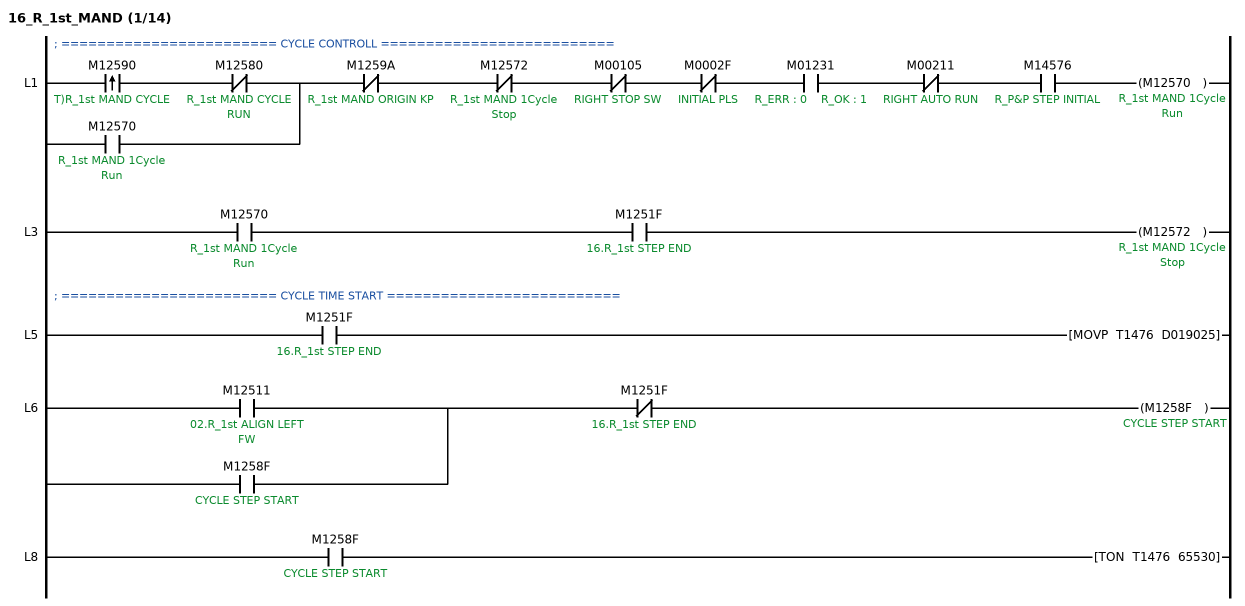
// ======================== CYCLE CONTROLL ==========================
; L1
LOADP     M12590	// T)R_1st MAND CYCLE
AND NOT   M12580	// R_1st MAND CYCLE RUN
OR        M12570	// R_1st MAND 1Cycle Run
AND NOT   M1259A	// R_1st MAND ORIGIN KP
AND NOT   M12572	// R_1st MAND 1Cycle Stop
AND NOT   M00105	// RIGHT STOP SW
AND NOT   M0002F	// INITIAL PLS
AND       M01231	// R_ERR : 0    R_OK : 1
AND NOT   M00211	// RIGHT AUTO RUN
AND       M14576	// R_P&P STEP INITIAL
OUT       M12570	// R_1st MAND 1Cycle Run
; L3
LOAD      M12570	// R_1st MAND 1Cycle Run
AND       M1251F	// 16.R_1st STEP END
OUT       M12572	// R_1st MAND 1Cycle Stop
// ======================== CYCLE TIME START ==========================
; L5
LOAD      M1251F	// 16.R_1st STEP END
MOVP      T1476 D019025
; L6
LOAD      M12511	// 02.R_1st ALIGN LEFT FW
OR        M1258F	// CYCLE STEP START
AND NOT   M1251F	// 16.R_1st STEP END
OUT       M1258F	// CYCLE STEP START
; L8
LOAD      M1258F	// CYCLE STEP START
TON       T1476 65530

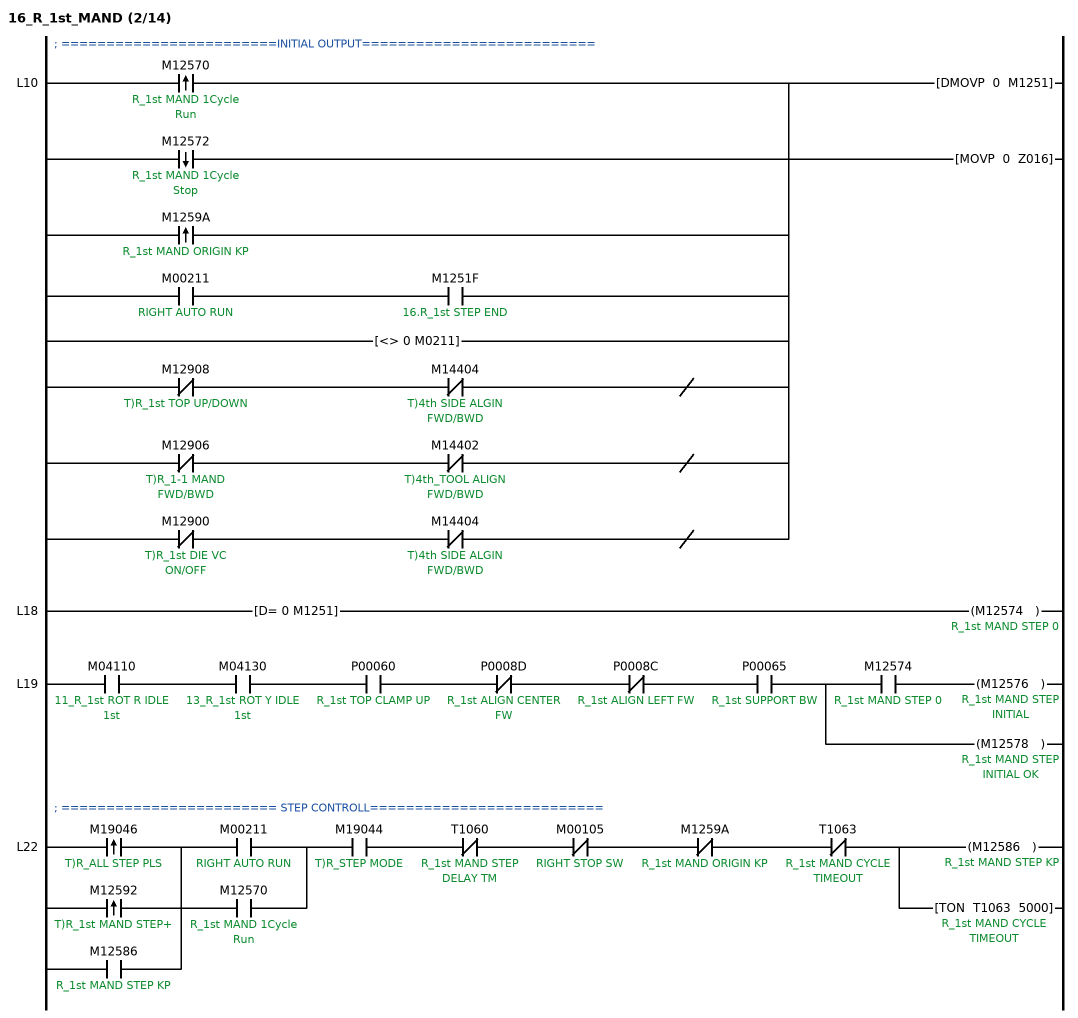
// ========================INITIAL OUTPUT==========================
; L10
LOADP     M12570	// R_1st MAND 1Cycle Run
ORN       M12572	// R_1st MAND 1Cycle Stop
ORP       M1259A	// R_1st MAND ORIGIN KP
LOAD      M00211	// RIGHT AUTO RUN
AND       M1251F	// 16.R_1st STEP END
OR LOAD
OR<>      0 M0211
LOAD NOT  M12908	// T)R_1st TOP UP/DOWN
AND NOT   M14404	// T)4th SIDE ALGIN FWD/BWD
NOT
OR LOAD
LOAD NOT  M12906	// T)R_1-1 MAND FWD/BWD
AND NOT   M14402	// T)4th_TOOL ALIGN FWD/BWD
NOT
OR LOAD
LOAD NOT  M12900	// T)R_1st DIE VC ON/OFF
AND NOT   M14404	// T)4th SIDE ALGIN FWD/BWD
NOT
OR LOAD
DMOVP     0 M1251
MOVP      0 Z016
; L18
LOADD=    0 M1251
OUT       M12574	// R_1st MAND STEP 0
; L19
LOAD      M04110	// 11_R_1st ROT R IDLE 1st
AND       M04130	// 13_R_1st ROT Y IDLE 1st
AND       P00060	// R_1st TOP CLAMP UP
AND NOT   P0008D	// R_1st ALIGN CENTER FW
AND NOT   P0008C	// R_1st ALIGN LEFT FW
AND       P00065	// R_1st SUPPORT BW
MPUSH
AND       M12574	// R_1st MAND STEP 0
OUT       M12576	// R_1st MAND STEP INITIAL
MPOP
OUT       M12578	// R_1st MAND STEP INITIAL OK
// ======================== STEP CONTROLL==========================
; L22
LOADP     M19046	// T)R_ALL STEP PLS
ORP       M12592	// T)R_1st MAND STEP+
OR        M12586	// R_1st MAND STEP KP
LOAD      M00211	// RIGHT AUTO RUN
OR        M12570	// R_1st MAND 1Cycle Run
AND LOAD
AND       M19044	// T)R_STEP MODE
AND NOT   T1060	// R_1st MAND STEP DELAY TM
AND NOT   M00105	// RIGHT STOP SW
AND NOT   M1259A	// R_1st MAND ORIGIN KP
AND NOT   T1063	// R_1st MAND CYCLE TIMEOUT
OUT       M12586	// R_1st MAND STEP KP
TON       T1063 5000	// R_1st MAND CYCLE TIMEOUT

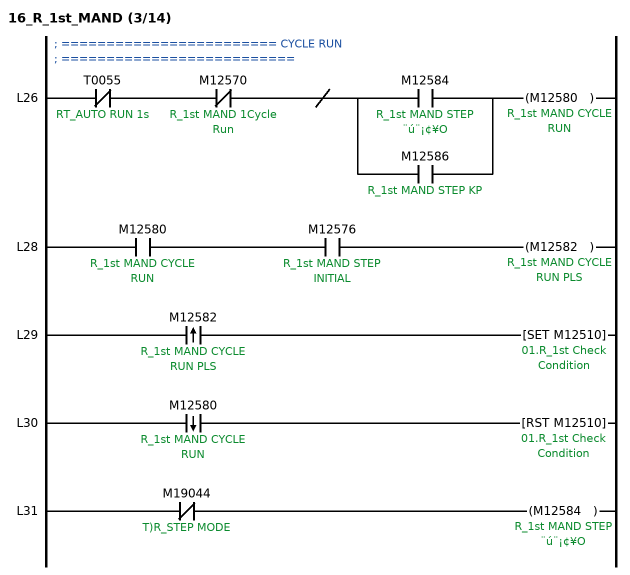
// ======================== CYCLE RUN ==========================
; L26
LOAD NOT  T0055	// RT_AUTO RUN 1s
AND NOT   M12570	// R_1st MAND 1Cycle Run
NOT
LOAD      M12584	// R_1st MAND STEP ¨ú¨¡¢¥O
OR        M12586	// R_1st MAND STEP KP
AND LOAD
OUT       M12580	// R_1st MAND CYCLE RUN
; L28
LOAD      M12580	// R_1st MAND CYCLE RUN
AND       M12576	// R_1st MAND STEP INITIAL
OUT       M12582	// R_1st MAND CYCLE RUN PLS
; L29
LOADP     M12582	// R_1st MAND CYCLE RUN PLS
SET       M12510	// 01.R_1st Check Condition
; L30
LOADN     M12580	// R_1st MAND CYCLE RUN
RST       M12510	// 01.R_1st Check Condition
; L31
LOAD NOT  M19044	// T)R_STEP MODE
OUT       M12584	// R_1st MAND STEP ¨ú¨¡¢¥O

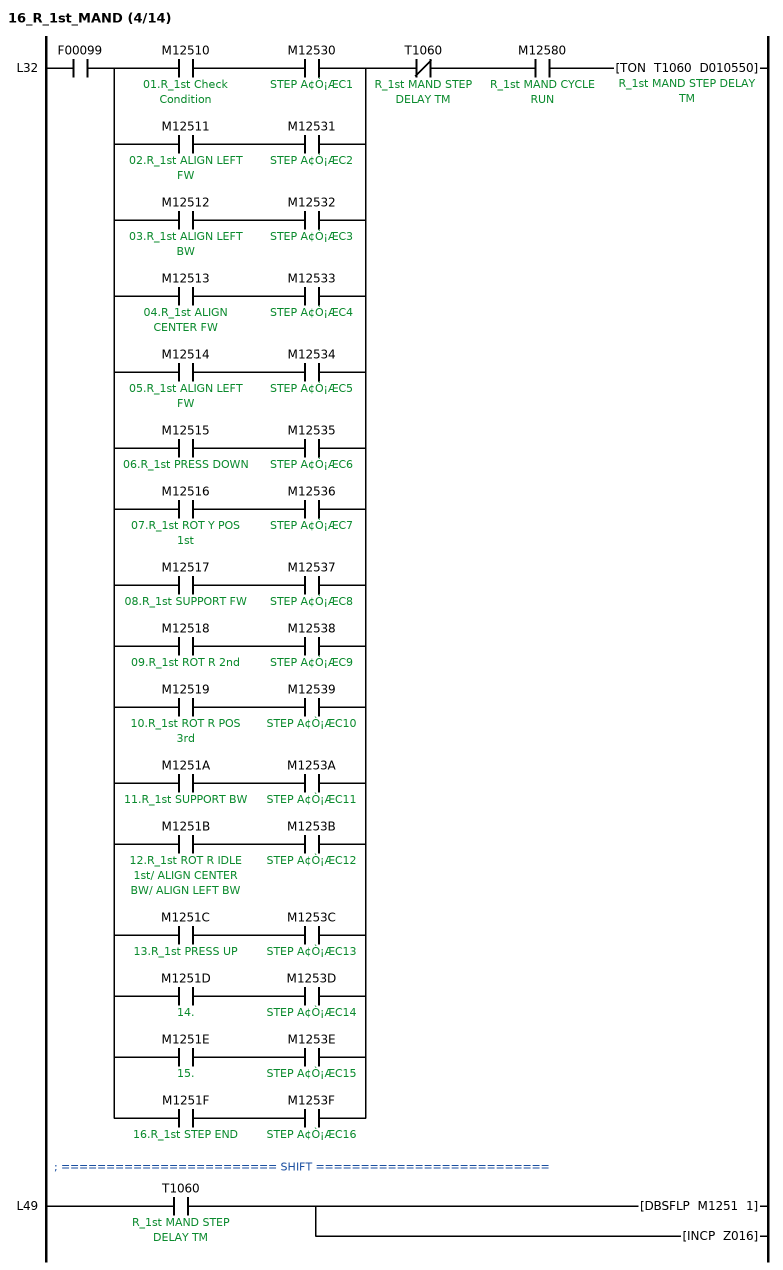
; L32
LOAD      F00099
LOAD      M12510	// 01.R_1st Check Condition
AND       M12530	// STEP A¢Ò¡ÆC1
LOAD      M12511	// 02.R_1st ALIGN LEFT FW
AND       M12531	// STEP A¢Ò¡ÆC2
OR LOAD
LOAD      M12512	// 03.R_1st ALIGN LEFT BW
AND       M12532	// STEP A¢Ò¡ÆC3
OR LOAD
LOAD      M12513	// 04.R_1st ALIGN CENTER FW
AND       M12533	// STEP A¢Ò¡ÆC4
OR LOAD
LOAD      M12514	// 05.R_1st ALIGN LEFT FW
AND       M12534	// STEP A¢Ò¡ÆC5
OR LOAD
LOAD      M12515	// 06.R_1st PRESS DOWN
AND       M12535	// STEP A¢Ò¡ÆC6
OR LOAD
LOAD      M12516	// 07.R_1st ROT Y POS 1st
AND       M12536	// STEP A¢Ò¡ÆC7
OR LOAD
LOAD      M12517	// 08.R_1st SUPPORT FW
AND       M12537	// STEP A¢Ò¡ÆC8
OR LOAD
LOAD      M12518	// 09.R_1st ROT R 2nd
AND       M12538	// STEP A¢Ò¡ÆC9
OR LOAD
LOAD      M12519	// 10.R_1st ROT R POS 3rd
AND       M12539	// STEP A¢Ò¡ÆC10
OR LOAD
LOAD      M1251A	// 11.R_1st SUPPORT BW
AND       M1253A	// STEP A¢Ò¡ÆC11
OR LOAD
LOAD      M1251B	// 12.R_1st ROT R IDLE 1st/ ALIGN CENTER BW/ ALIGN LEFT BW
AND       M1253B	// STEP A¢Ò¡ÆC12
OR LOAD
LOAD      M1251C	// 13.R_1st PRESS UP
AND       M1253C	// STEP A¢Ò¡ÆC13
OR LOAD
LOAD      M1251D	// 14.
AND       M1253D	// STEP A¢Ò¡ÆC14
OR LOAD
LOAD      M1251E	// 15.
AND       M1253E	// STEP A¢Ò¡ÆC15
OR LOAD
LOAD      M1251F	// 16.R_1st STEP END
AND       M1253F	// STEP A¢Ò¡ÆC16
OR LOAD
AND LOAD
AND NOT   T1060	// R_1st MAND STEP DELAY TM
AND       M12580	// R_1st MAND CYCLE RUN
TON       T1060 D010550	// R_1st MAND STEP DELAY TM
// ======================== SHIFT ==========================
; L49
LOAD      T1060	// R_1st MAND STEP DELAY TM
DBSFLP    M1251 1
INCP      Z016

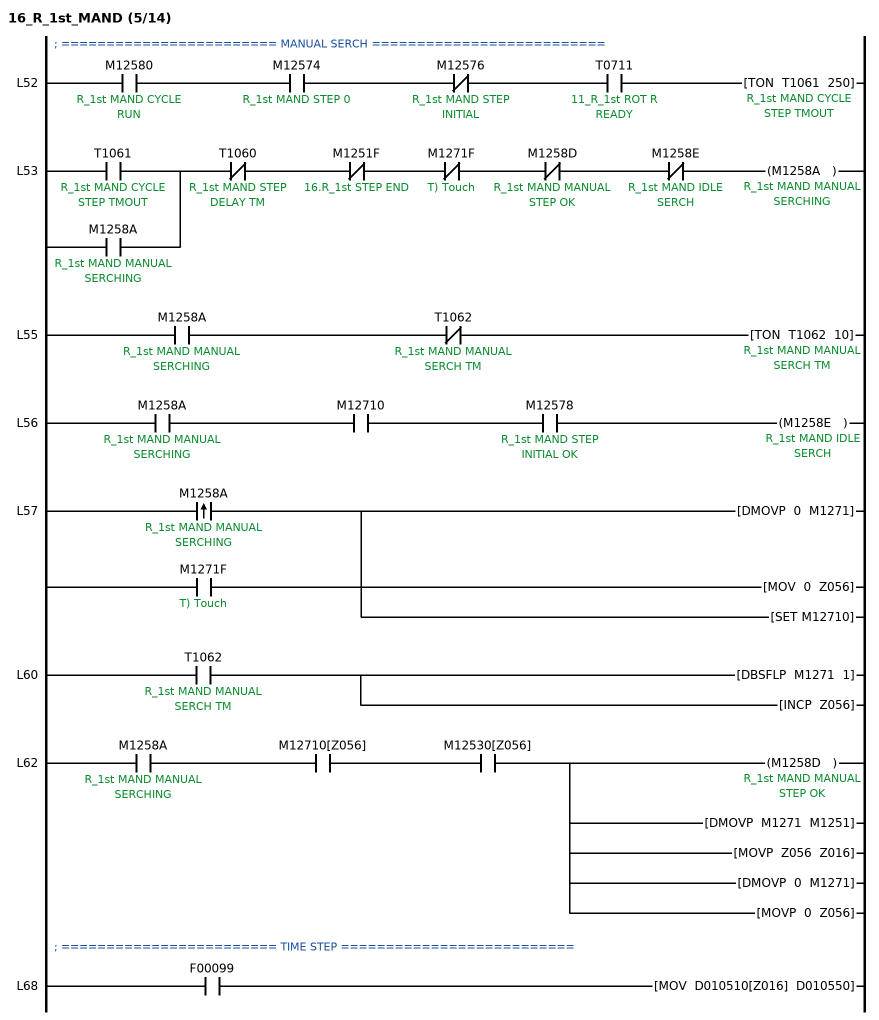
// ======================== MANUAL SERCH ==========================
; L52
LOAD      M12580	// R_1st MAND CYCLE RUN
AND       M12574	// R_1st MAND STEP 0
AND NOT   M12576	// R_1st MAND STEP INITIAL
AND       T0711	// 11_R_1st ROT R READY
TON       T1061 250	// R_1st MAND CYCLE STEP TMOUT
; L53
LOAD      T1061	// R_1st MAND CYCLE STEP TMOUT
OR        M1258A	// R_1st MAND MANUAL SERCHING
AND NOT   T1060	// R_1st MAND STEP DELAY TM
AND NOT   M1251F	// 16.R_1st STEP END
AND NOT   M1271F	// T) Touch
AND NOT   M1258D	// R_1st MAND MANUAL STEP OK
AND NOT   M1258E	// R_1st MAND IDLE SERCH
OUT       M1258A	// R_1st MAND MANUAL SERCHING
; L55
LOAD      M1258A	// R_1st MAND MANUAL SERCHING
AND NOT   T1062	// R_1st MAND MANUAL SERCH TM
TON       T1062 10	// R_1st MAND MANUAL SERCH TM
; L56
LOAD      M1258A	// R_1st MAND MANUAL SERCHING
AND       M12710
AND       M12578	// R_1st MAND STEP INITIAL OK
OUT       M1258E	// R_1st MAND IDLE SERCH
; L57
LOADP     M1258A	// R_1st MAND MANUAL SERCHING
OR        M1271F	// T) Touch
DMOVP     0 M1271
MOV       0 Z056
SET       M12710
; L60
LOAD      T1062	// R_1st MAND MANUAL SERCH TM
DBSFLP    M1271 1
INCP      Z056
; L62
LOAD      M1258A	// R_1st MAND MANUAL SERCHING
AND       M12710[Z056]
AND       M12530[Z056]
OUT       M1258D	// R_1st MAND MANUAL STEP OK
DMOVP     M1271 M1251
MOVP      Z056 Z016
DMOVP     0 M1271
MOVP      0 Z056
// ======================== TIME STEP ==========================
; L68
LOAD      F00099
MOV       D010510[Z016] D010550

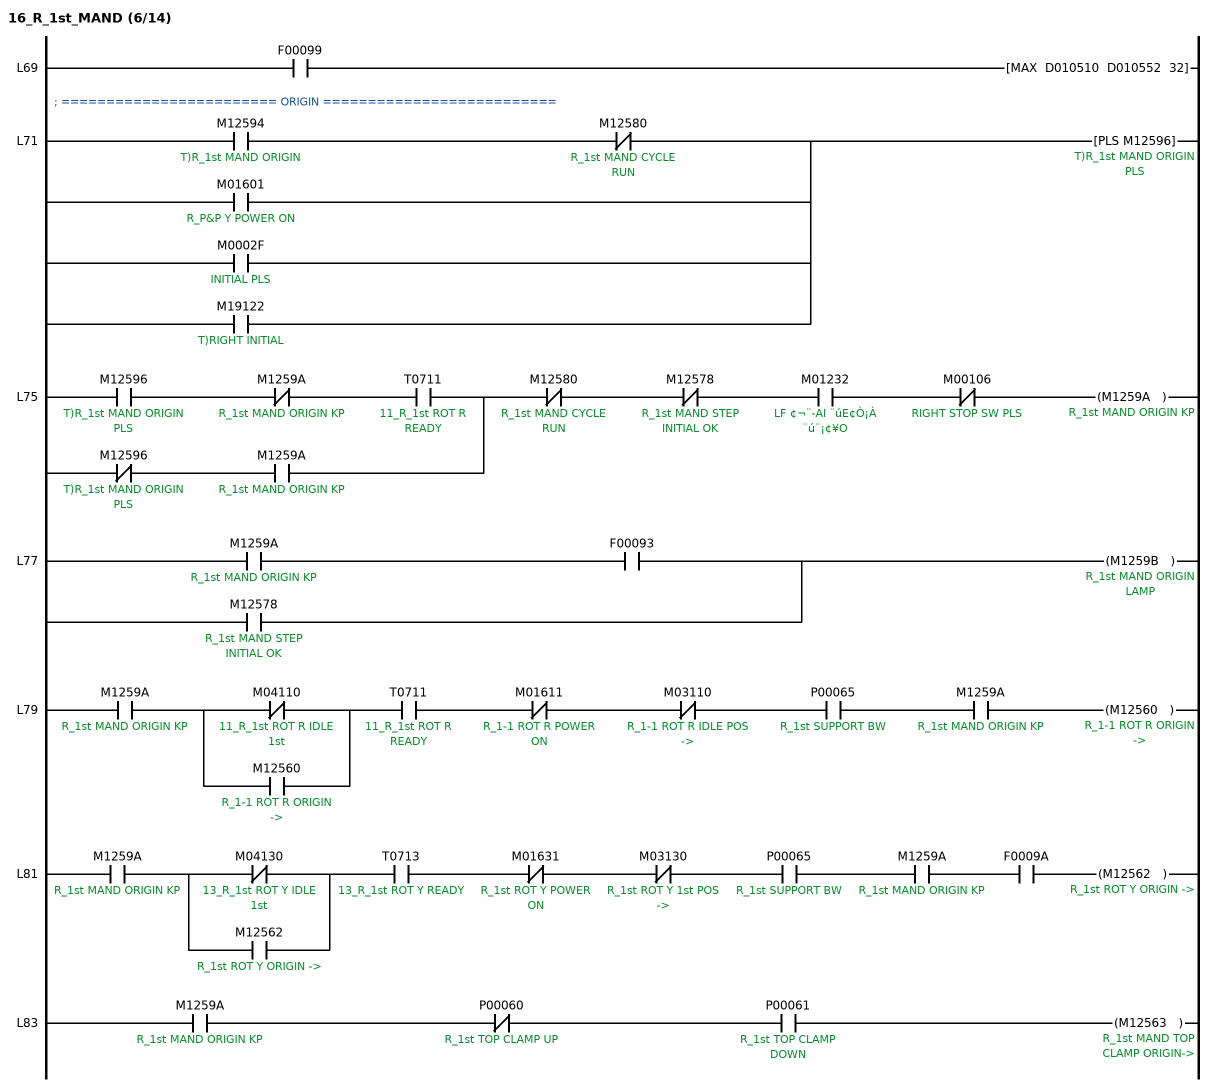
; L69
LOAD      F00099
MAX       D010510 D010552 32
// ======================== ORIGIN ==========================
; L71
LOAD      M12594	// T)R_1st MAND ORIGIN
AND NOT   M12580	// R_1st MAND CYCLE RUN
OR        M01601	// R_P&P Y POWER ON
OR        M0002F	// INITIAL PLS
OR        M19122	// T)RIGHT INITIAL
OUTP      M12596	// T)R_1st MAND ORIGIN PLS
; L75
LOAD      M12596	// T)R_1st MAND ORIGIN PLS
AND NOT   M1259A	// R_1st MAND ORIGIN KP
AND       T0711	// 11_R_1st ROT R READY
LOAD NOT  M12596	// T)R_1st MAND ORIGIN PLS
AND       M1259A	// R_1st MAND ORIGIN KP
OR LOAD
AND NOT   M12580	// R_1st MAND CYCLE RUN
AND NOT   M12578	// R_1st MAND STEP INITIAL OK
AND       M01232	// LF ¢¬¨­AI ¨úE¢Ò¡À ¨ú¨¡¢¥O
AND NOT   M00106	// RIGHT STOP SW PLS
OUT       M1259A	// R_1st MAND ORIGIN KP
; L77
LOAD      M1259A	// R_1st MAND ORIGIN KP
AND       F00093
OR        M12578	// R_1st MAND STEP INITIAL OK
OUT       M1259B	// R_1st MAND ORIGIN LAMP
; L79
LOAD      M1259A	// R_1st MAND ORIGIN KP
LOAD NOT  M04110	// 11_R_1st ROT R IDLE 1st
OR        M12560	// R_1-1 ROT R ORIGIN ->
AND LOAD
AND       T0711	// 11_R_1st ROT R READY
AND NOT   M01611	// R_1-1 ROT R POWER ON
AND NOT   M03110	// R_1-1 ROT R IDLE POS ->
AND       P00065	// R_1st SUPPORT BW
AND       M1259A	// R_1st MAND ORIGIN KP
OUT       M12560	// R_1-1 ROT R ORIGIN ->
; L81
LOAD      M1259A	// R_1st MAND ORIGIN KP
LOAD NOT  M04130	// 13_R_1st ROT Y IDLE 1st
OR        M12562	// R_1st ROT Y ORIGIN ->
AND LOAD
AND       T0713	// 13_R_1st ROT Y READY
AND NOT   M01631	// R_1st ROT Y POWER ON
AND NOT   M03130	// R_1st ROT Y 1st POS ->
AND       P00065	// R_1st SUPPORT BW
AND       M1259A	// R_1st MAND ORIGIN KP
AND       F0009A
OUT       M12562	// R_1st ROT Y ORIGIN ->
; L83
LOAD      M1259A	// R_1st MAND ORIGIN KP
AND NOT   P00060	// R_1st TOP CLAMP UP
AND       P00061	// R_1st TOP CLAMP DOWN
OUT       M12563	// R_1st MAND TOP CLAMP ORIGIN->

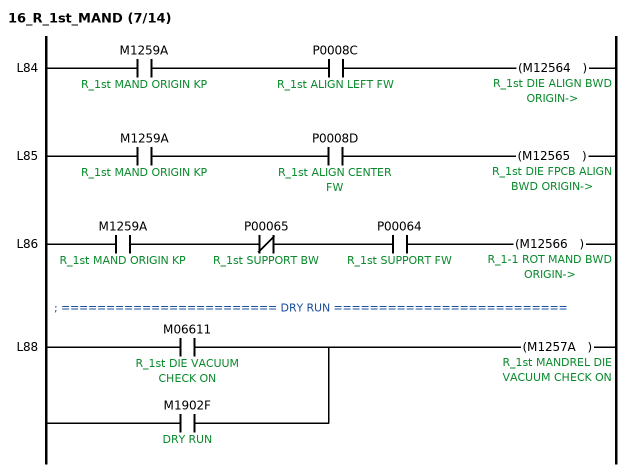
; L84
LOAD      M1259A	// R_1st MAND ORIGIN KP
AND       P0008C	// R_1st ALIGN LEFT FW
OUT       M12564	// R_1st DIE ALIGN BWD ORIGIN->
; L85
LOAD      M1259A	// R_1st MAND ORIGIN KP
AND       P0008D	// R_1st ALIGN CENTER FW
OUT       M12565	// R_1st DIE FPCB ALIGN BWD ORIGIN->
; L86
LOAD      M1259A	// R_1st MAND ORIGIN KP
AND NOT   P00065	// R_1st SUPPORT BW
AND       P00064	// R_1st SUPPORT FW
OUT       M12566	// R_1-1 ROT MAND BWD ORIGIN->
// ======================== DRY RUN ==========================
; L88
LOAD      M06611	// R_1st DIE VACUUM CHECK ON
OR        M1902F	// DRY RUN
OUT       M1257A	// R_1st MANDREL DIE VACUUM CHECK ON

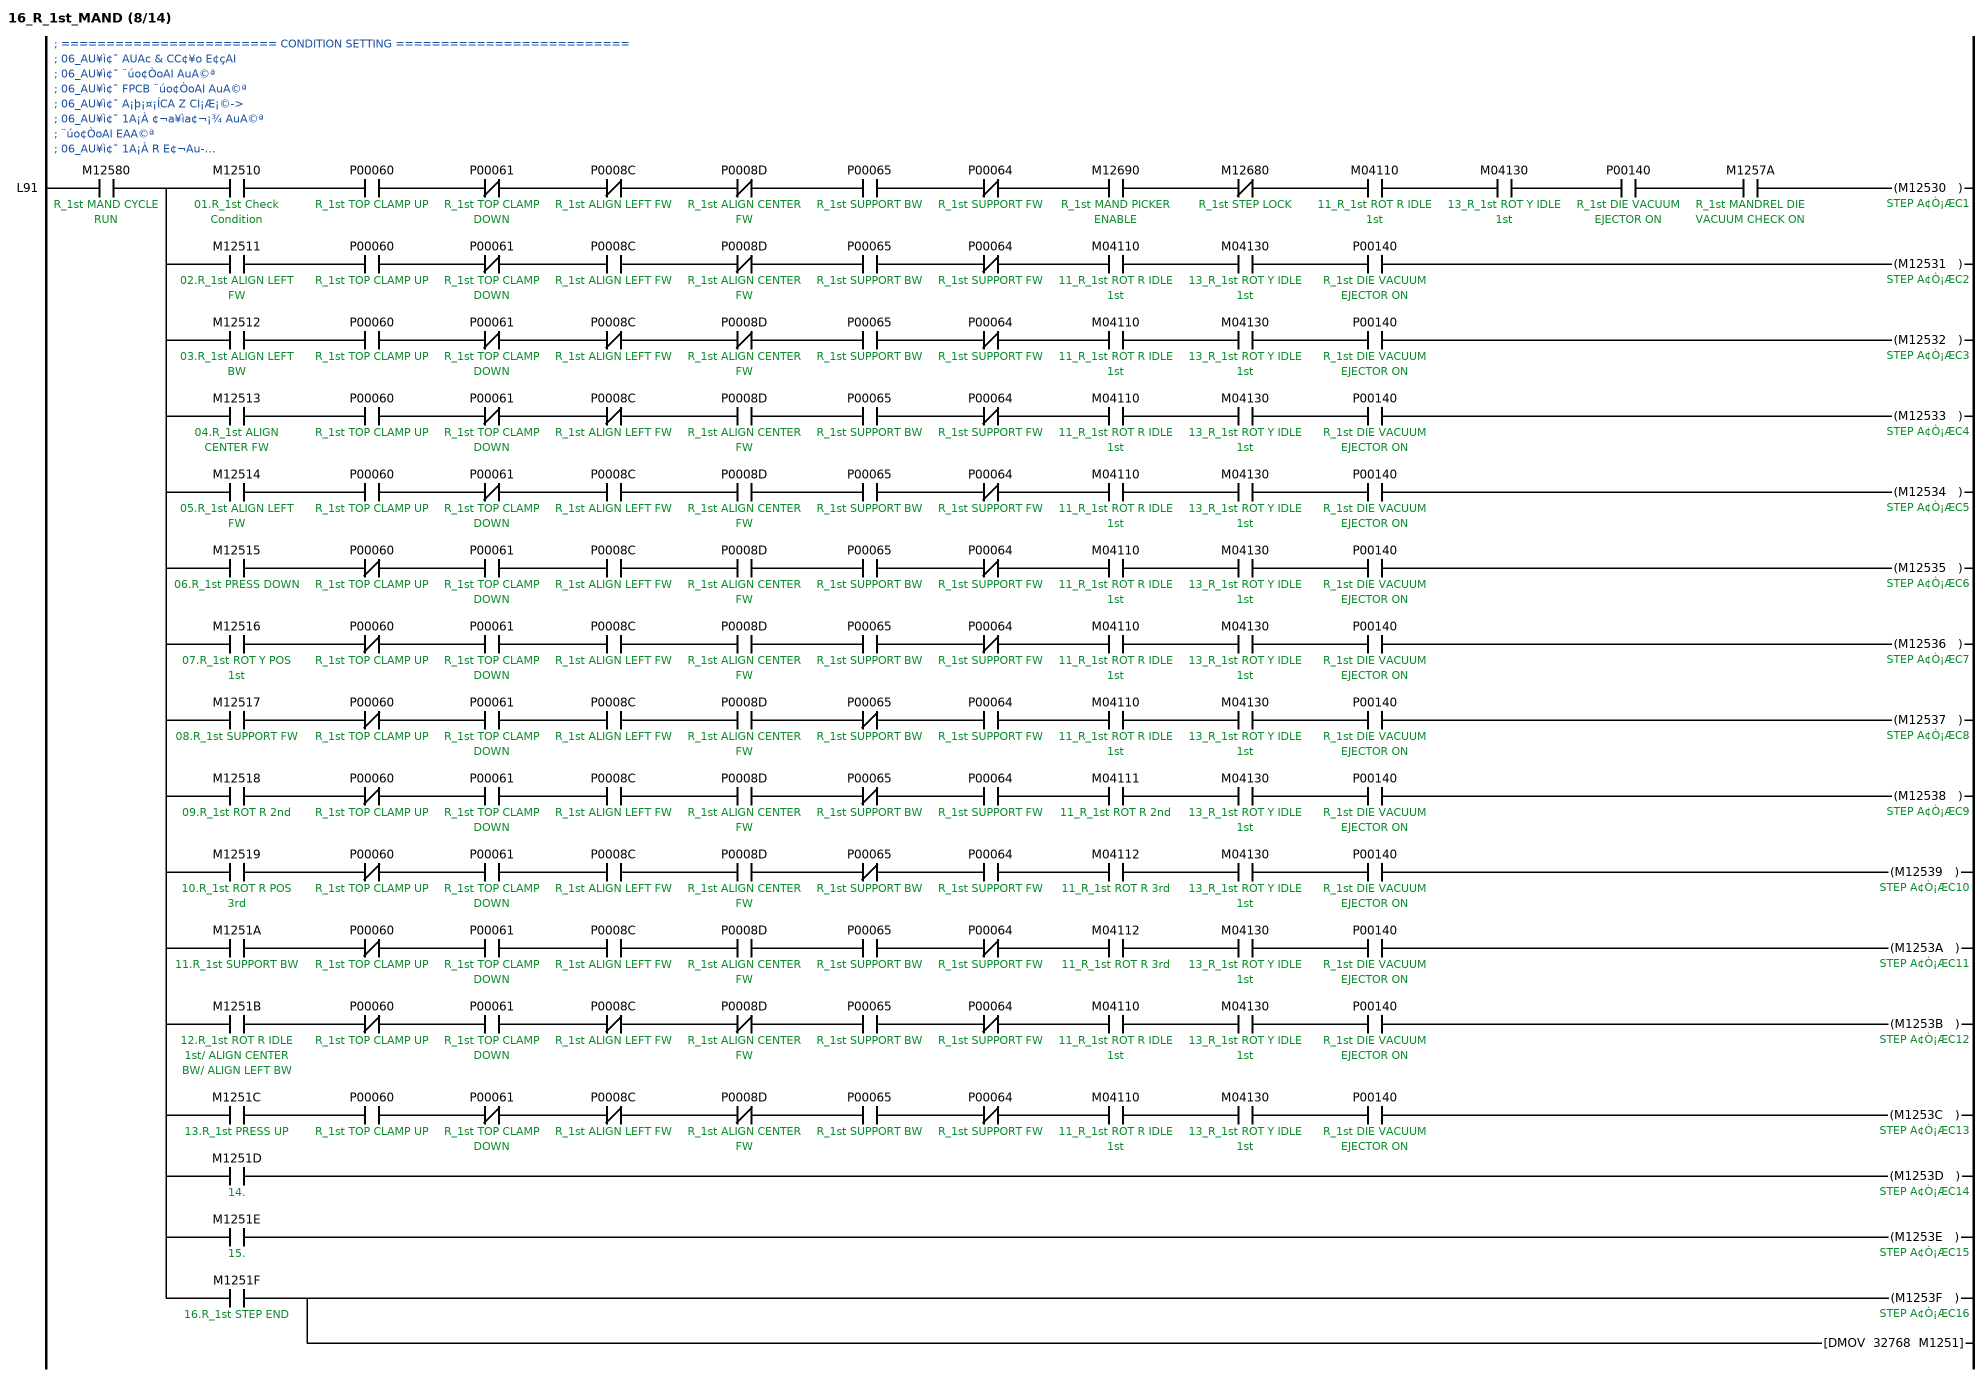
// ======================== CONDITION SETTING ==========================
; L91
LOAD      M12580	// R_1st MAND CYCLE RUN
MPUSH
AND       M12510	// 01.R_1st Check Condition
AND       P00060	// R_1st TOP CLAMP UP
AND NOT   P00061	// R_1st TOP CLAMP DOWN
AND NOT   P0008C	// R_1st ALIGN LEFT FW
AND NOT   P0008D	// R_1st ALIGN CENTER FW
AND       P00065	// R_1st SUPPORT BW
AND NOT   P00064	// R_1st SUPPORT FW
AND       M12690	// R_1st MAND PICKER ENABLE
AND NOT   M12680	// R_1st STEP LOCK
AND       M04110	// 11_R_1st ROT R IDLE 1st
AND       M04130	// 13_R_1st ROT Y IDLE 1st
AND       P00140	// R_1st DIE VACUUM EJECTOR ON
AND       M1257A	// R_1st MANDREL DIE VACUUM CHECK ON
OUT       M12530	// STEP A¢Ò¡ÆC1
MLOAD
AND       M12511	// 02.R_1st ALIGN LEFT FW
AND       P00060	// R_1st TOP CLAMP UP
AND NOT   P00061	// R_1st TOP CLAMP DOWN
AND       P0008C	// R_1st ALIGN LEFT FW
AND NOT   P0008D	// R_1st ALIGN CENTER FW
AND       P00065	// R_1st SUPPORT BW
AND NOT   P00064	// R_1st SUPPORT FW
AND       M04110	// 11_R_1st ROT R IDLE 1st
AND       M04130	// 13_R_1st ROT Y IDLE 1st
AND       P00140	// R_1st DIE VACUUM EJECTOR ON
OUT       M12531	// STEP A¢Ò¡ÆC2
MLOAD
AND       M12512	// 03.R_1st ALIGN LEFT BW
AND       P00060	// R_1st TOP CLAMP UP
AND NOT   P00061	// R_1st TOP CLAMP DOWN
AND NOT   P0008C	// R_1st ALIGN LEFT FW
AND NOT   P0008D	// R_1st ALIGN CENTER FW
AND       P00065	// R_1st SUPPORT BW
AND NOT   P00064	// R_1st SUPPORT FW
AND       M04110	// 11_R_1st ROT R IDLE 1st
AND       M04130	// 13_R_1st ROT Y IDLE 1st
AND       P00140	// R_1st DIE VACUUM EJECTOR ON
OUT       M12532	// STEP A¢Ò¡ÆC3
MLOAD
AND       M12513	// 04.R_1st ALIGN CENTER FW
AND       P00060	// R_1st TOP CLAMP UP
AND NOT   P00061	// R_1st TOP CLAMP DOWN
AND NOT   P0008C	// R_1st ALIGN LEFT FW
AND       P0008D	// R_1st ALIGN CENTER FW
AND       P00065	// R_1st SUPPORT BW
AND NOT   P00064	// R_1st SUPPORT FW
AND       M04110	// 11_R_1st ROT R IDLE 1st
AND       M04130	// 13_R_1st ROT Y IDLE 1st
AND       P00140	// R_1st DIE VACUUM EJECTOR ON
OUT       M12533	// STEP A¢Ò¡ÆC4
MLOAD
AND       M12514	// 05.R_1st ALIGN LEFT FW
AND       P00060	// R_1st TOP CLAMP UP
AND NOT   P00061	// R_1st TOP CLAMP DOWN
AND       P0008C	// R_1st ALIGN LEFT FW
AND       P0008D	// R_1st ALIGN CENTER FW
AND       P00065	// R_1st SUPPORT BW
AND NOT   P00064	// R_1st SUPPORT FW
AND       M04110	// 11_R_1st ROT R IDLE 1st
AND       M04130	// 13_R_1st ROT Y IDLE 1st
AND       P00140	// R_1st DIE VACUUM EJECTOR ON
OUT       M12534	// STEP A¢Ò¡ÆC5
MLOAD
AND       M12515	// 06.R_1st PRESS DOWN
AND NOT   P00060	// R_1st TOP CLAMP UP
AND       P00061	// R_1st TOP CLAMP DOWN
AND       P0008C	// R_1st ALIGN LEFT FW
AND       P0008D	// R_1st ALIGN CENTER FW
AND       P00065	// R_1st SUPPORT BW
AND NOT   P00064	// R_1st SUPPORT FW
AND       M04110	// 11_R_1st ROT R IDLE 1st
AND       M04130	// 13_R_1st ROT Y IDLE 1st
AND       P00140	// R_1st DIE VACUUM EJECTOR ON
OUT       M12535	// STEP A¢Ò¡ÆC6
MLOAD
AND       M12516	// 07.R_1st ROT Y POS 1st
AND NOT   P00060	// R_1st TOP CLAMP UP
AND       P00061	// R_1st TOP CLAMP DOWN
AND       P0008C	// R_1st ALIGN LEFT FW
AND       P0008D	// R_1st ALIGN CENTER FW
AND       P00065	// R_1st SUPPORT BW
AND NOT   P00064	// R_1st SUPPORT FW
AND       M04110	// 11_R_1st ROT R IDLE 1st
AND       M04130	// 13_R_1st ROT Y IDLE 1st
AND       P00140	// R_1st DIE VACUUM EJECTOR ON
OUT       M12536	// STEP A¢Ò¡ÆC7
MLOAD
AND       M12517	// 08.R_1st SUPPORT FW
AND NOT   P00060	// R_1st TOP CLAMP UP
AND       P00061	// R_1st TOP CLAMP DOWN
AND       P0008C	// R_1st ALIGN LEFT FW
AND       P0008D	// R_1st ALIGN CENTER FW
AND NOT   P00065	// R_1st SUPPORT BW
AND       P00064	// R_1st SUPPORT FW
AND       M04110	// 11_R_1st ROT R IDLE 1st
AND       M04130	// 13_R_1st ROT Y IDLE 1st
AND       P00140	// R_1st DIE VACUUM EJECTOR ON
OUT       M12537	// STEP A¢Ò¡ÆC8
MLOAD
AND       M12518	// 09.R_1st ROT R 2nd
AND NOT   P00060	// R_1st TOP CLAMP UP
AND       P00061	// R_1st TOP CLAMP DOWN
AND       P0008C	// R_1st ALIGN LEFT FW
AND       P0008D	// R_1st ALIGN CENTER FW
AND NOT   P00065	// R_1st SUPPORT BW
AND       P00064	// R_1st SUPPORT FW
AND       M04111	// 11_R_1st ROT R 2nd
AND       M04130	// 13_R_1st ROT Y IDLE 1st
AND       P00140	// R_1st DIE VACUUM EJECTOR ON
OUT       M12538	// STEP A¢Ò¡ÆC9
MLOAD
AND       M12519	// 10.R_1st ROT R POS 3rd
AND NOT   P00060	// R_1st TOP CLAMP UP
AND       P00061	// R_1st TOP CLAMP DOWN
AND       P0008C	// R_1st ALIGN LEFT FW
AND       P0008D	// R_1st ALIGN CENTER FW
AND NOT   P00065	// R_1st SUPPORT BW
AND       P00064	// R_1st SUPPORT FW
AND       M04112	// 11_R_1st ROT R 3rd
AND       M04130	// 13_R_1st ROT Y IDLE 1st
AND       P00140	// R_1st DIE VACUUM EJECTOR ON
OUT       M12539	// STEP A¢Ò¡ÆC10
MLOAD
AND       M1251A	// 11.R_1st SUPPORT BW
AND NOT   P00060	// R_1st TOP CLAMP UP
AND       P00061	// R_1st TOP CLAMP DOWN
AND       P0008C	// R_1st ALIGN LEFT FW
AND       P0008D	// R_1st ALIGN CENTER FW
AND       P00065	// R_1st SUPPORT BW
AND NOT   P00064	// R_1st SUPPORT FW
AND       M04112	// 11_R_1st ROT R 3rd
AND       M04130	// 13_R_1st ROT Y IDLE 1st
AND       P00140	// R_1st DIE VACUUM EJECTOR ON
OUT       M1253A	// STEP A¢Ò¡ÆC11
MLOAD
AND       M1251B	// 12.R_1st ROT R IDLE 1st/ ALIGN CENTER BW/ ALIGN LEFT BW
AND NOT   P00060	// R_1st TOP CLAMP UP
AND       P00061	// R_1st TOP CLAMP DOWN
AND NOT   P0008C	// R_1st ALIGN LEFT FW
AND NOT   P0008D	// R_1st ALIGN CENTER FW
AND       P00065	// R_1st SUPPORT BW
AND NOT   P00064	// R_1st SUPPORT FW
AND       M04110	// 11_R_1st ROT R IDLE 1st
AND       M04130	// 13_R_1st ROT Y IDLE 1st
AND       P00140	// R_1st DIE VACUUM EJECTOR ON
OUT       M1253B	// STEP A¢Ò¡ÆC12
MLOAD
AND       M1251C	// 13.R_1st PRESS UP
AND       P00060	// R_1st TOP CLAMP UP
AND NOT   P00061	// R_1st TOP CLAMP DOWN
AND NOT   P0008C	// R_1st ALIGN LEFT FW
AND NOT   P0008D	// R_1st ALIGN CENTER FW
AND       P00065	// R_1st SUPPORT BW
AND NOT   P00064	// R_1st SUPPORT FW
AND       M04110	// 11_R_1st ROT R IDLE 1st
AND       M04130	// 13_R_1st ROT Y IDLE 1st
AND       P00140	// R_1st DIE VACUUM EJECTOR ON
OUT       M1253C	// STEP A¢Ò¡ÆC13
MLOAD
AND       M1251D	// 14.
OUT       M1253D	// STEP A¢Ò¡ÆC14
MLOAD
AND       M1251E	// 15.
OUT       M1253E	// STEP A¢Ò¡ÆC15
MPOP
AND       M1251F	// 16.R_1st STEP END
OUT       M1253F	// STEP A¢Ò¡ÆC16
DMOV      32768 M1251
// output comment: 06_AU¥ì¢¯ AUAc & CC¢¥o E¢çAI
// output comment: 06_AU¥ì¢¯ ¨úo¢ÒoAI AuA©ª
// output comment: 06_AU¥ì¢¯ FPCB ¨úo¢ÒoAI AuA©ª
// output comment: 06_AU¥ì¢¯ A¡þ¡¤¡ÍCA Z CI¡Æ¡©->
// output comment: 06_AU¥ì¢¯ 1A¡À ¢¬a¥ìa¢¬¡¾ AuA©ª ¨úo¢ÒoAI EAA©ª
// output comment: 06_AU¥ì¢¯ 1A¡À R E¢¬Au->
// output comment: 06_AU¥ì¢¯ 1A¡À R ¨¬©ö¡¾I->
// output comment: 06_AU¥ì¢¯ 1A¡À ¢¬a¥ìa¢¬¡¾ EAA©ª
// output comment: 06_AU¥ì¢¯ R ¢¥e¡¾a -> ¡ío¨¬I ¡ío¨öA

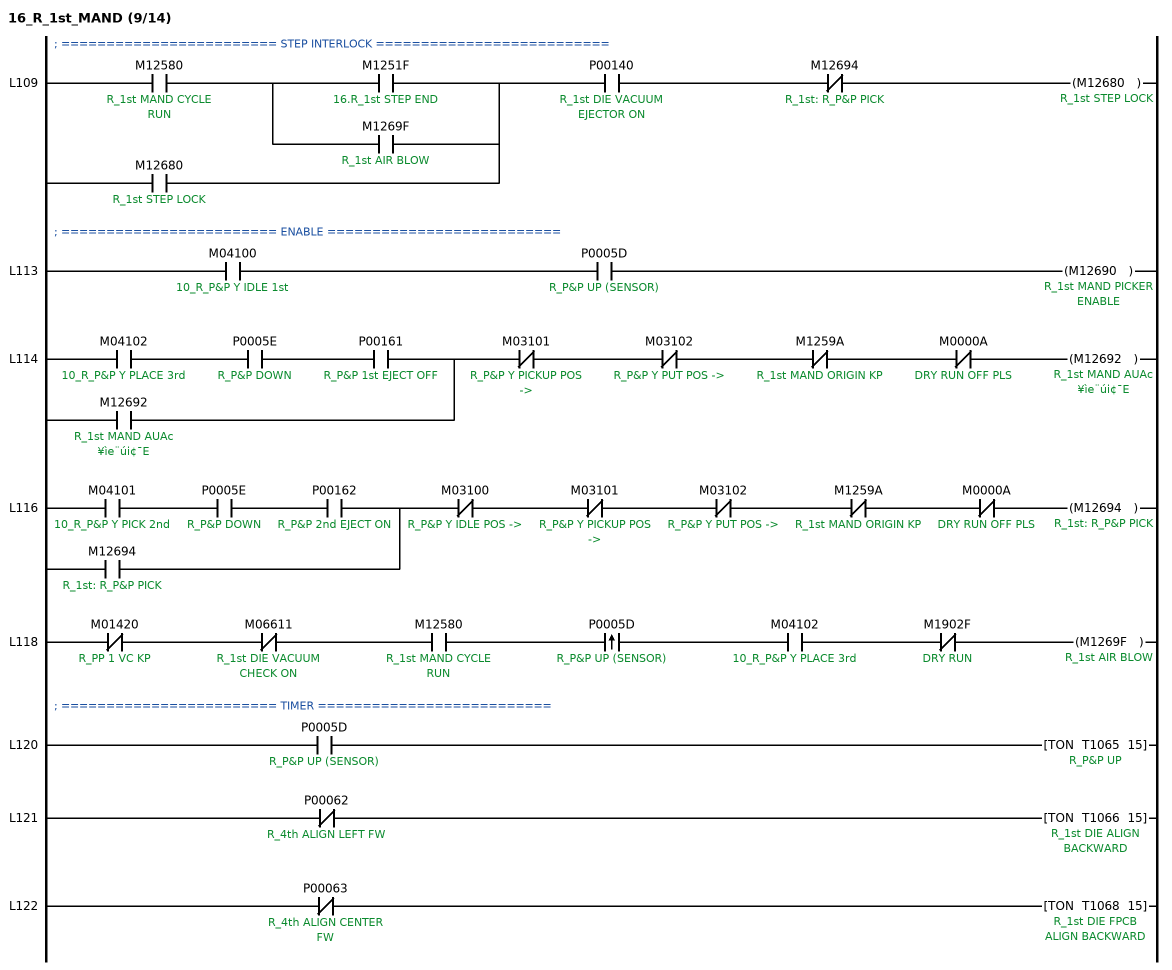
// ======================== STEP INTERLOCK ==========================
; L109
LOAD      M12580	// R_1st MAND CYCLE RUN
LOAD      M1251F	// 16.R_1st STEP END
OR        M1269F	// R_1st AIR BLOW
AND LOAD
OR        M12680	// R_1st STEP LOCK
AND       P00140	// R_1st DIE VACUUM EJECTOR ON
AND NOT   M12694	// R_1st: R_P&P PICK
OUT       M12680	// R_1st STEP LOCK
// ======================== ENABLE ==========================
; L113
LOAD      M04100	// 10_R_P&P Y IDLE 1st
AND       P0005D	// R_P&P UP (SENSOR)
OUT       M12690	// R_1st MAND PICKER ENABLE
; L114
LOAD      M04102	// 10_R_P&P Y PLACE 3rd
AND       P0005E	// R_P&P DOWN
AND       P00161	// R_P&P 1st EJECT OFF
OR        M12692	// R_1st MAND AUAc ¥ìe¨úi¢¯E
AND NOT   M03101	// R_P&P Y PICKUP POS ->
AND NOT   M03102	// R_P&P Y PUT POS ->
AND NOT   M1259A	// R_1st MAND ORIGIN KP
AND NOT   M0000A	// DRY RUN OFF PLS
OUT       M12692	// R_1st MAND AUAc ¥ìe¨úi¢¯E
; L116
LOAD      M04101	// 10_R_P&P Y PICK 2nd
AND       P0005E	// R_P&P DOWN
AND       P00162	// R_P&P 2nd EJECT ON
OR        M12694	// R_1st: R_P&P PICK
AND NOT   M03100	// R_P&P Y IDLE POS ->
AND NOT   M03101	// R_P&P Y PICKUP POS ->
AND NOT   M03102	// R_P&P Y PUT POS ->
AND NOT   M1259A	// R_1st MAND ORIGIN KP
AND NOT   M0000A	// DRY RUN OFF PLS
OUT       M12694	// R_1st: R_P&P PICK
; L118
LOAD NOT  M01420	// R_PP 1 VC KP
AND NOT   M06611	// R_1st DIE VACUUM CHECK ON
AND       M12580	// R_1st MAND CYCLE RUN
ANDP      P0005D	// R_P&P UP (SENSOR)
AND       M04102	// 10_R_P&P Y PLACE 3rd
AND NOT   M1902F	// DRY RUN
OUT       M1269F	// R_1st AIR BLOW
// ======================== TIMER ==========================
; L120
LOAD      P0005D	// R_P&P UP (SENSOR)
TON       T1065 15	// R_P&P UP
; L121
LOAD NOT  P00062	// R_4th ALIGN LEFT FW
TON       T1066 15	// R_1st DIE ALIGN BACKWARD
; L122
LOAD NOT  P00063	// R_4th ALIGN CENTER FW
TON       T1068 15	// R_1st DIE FPCB ALIGN BACKWARD

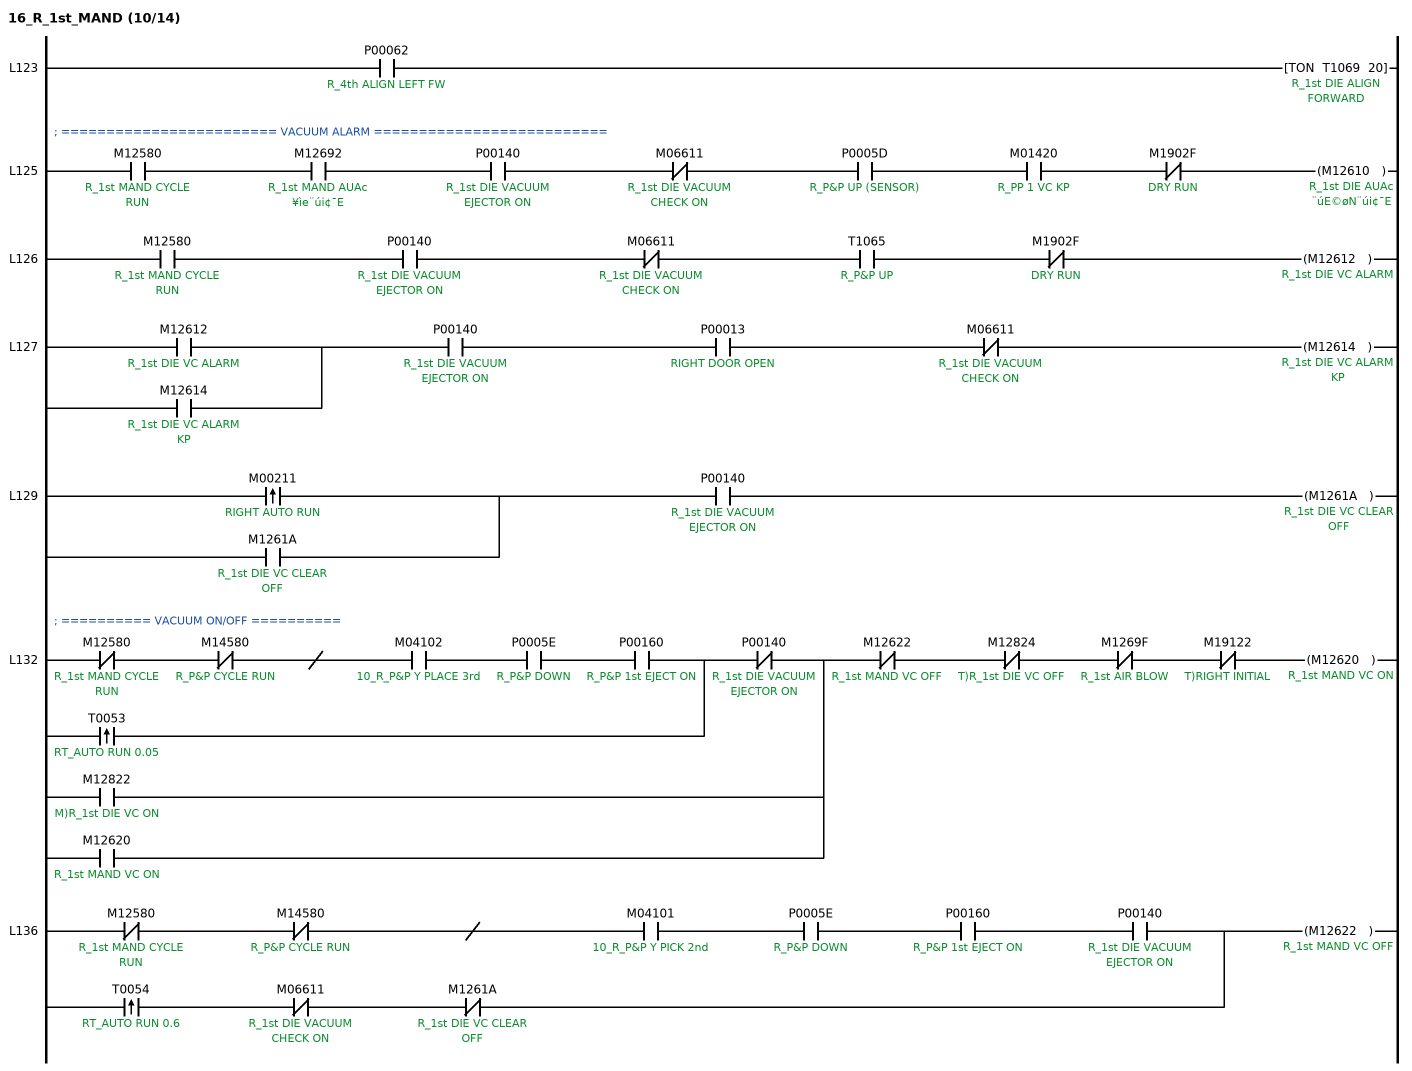
; L123
LOAD      P00062	// R_4th ALIGN LEFT FW
TON       T1069 20	// R_1st DIE ALIGN FORWARD
// ======================== VACUUM ALARM ==========================
; L125
LOAD      M12580	// R_1st MAND CYCLE RUN
AND       M12692	// R_1st MAND AUAc ¥ìe¨úi¢¯E
AND       P00140	// R_1st DIE VACUUM EJECTOR ON
AND NOT   M06611	// R_1st DIE VACUUM CHECK ON
AND       P0005D	// R_P&P UP (SENSOR)
AND       M01420	// R_PP 1 VC KP
AND NOT   M1902F	// DRY RUN
OUT       M12610	// R_1st DIE AUAc ¨úE©øN¨úi¢¯E
; L126
LOAD      M12580	// R_1st MAND CYCLE RUN
AND       P00140	// R_1st DIE VACUUM EJECTOR ON
AND NOT   M06611	// R_1st DIE VACUUM CHECK ON
AND       T1065	// R_P&P UP
AND NOT   M1902F	// DRY RUN
OUT       M12612	// R_1st DIE VC ALARM
; L127
LOAD      M12612	// R_1st DIE VC ALARM
OR        M12614	// R_1st DIE VC ALARM KP
AND       P00140	// R_1st DIE VACUUM EJECTOR ON
AND       P00013	// RIGHT DOOR OPEN
AND NOT   M06611	// R_1st DIE VACUUM CHECK ON
OUT       M12614	// R_1st DIE VC ALARM KP
; L129
LOADP     M00211	// RIGHT AUTO RUN
OR        M1261A	// R_1st DIE VC CLEAR OFF
AND       P00140	// R_1st DIE VACUUM EJECTOR ON
OUT       M1261A	// R_1st DIE VC CLEAR OFF
// ========== VACUUM ON/OFF ==========
; L132
LOAD NOT  M12580	// R_1st MAND CYCLE RUN
AND NOT   M14580	// R_P&P CYCLE RUN
NOT
AND       M04102	// 10_R_P&P Y PLACE 3rd
AND       P0005E	// R_P&P DOWN
AND       P00160	// R_P&P 1st EJECT ON
ORP       T0053	// RT_AUTO RUN 0.05
AND NOT   P00140	// R_1st DIE VACUUM EJECTOR ON
OR        M12822	// M)R_1st DIE VC ON
OR        M12620	// R_1st MAND VC ON
AND NOT   M12622	// R_1st MAND VC OFF
AND NOT   M12824	// T)R_1st DIE VC OFF
AND NOT   M1269F	// R_1st AIR BLOW
AND NOT   M19122	// T)RIGHT INITIAL
OUT       M12620	// R_1st MAND VC ON
; L136
LOAD NOT  M12580	// R_1st MAND CYCLE RUN
AND NOT   M14580	// R_P&P CYCLE RUN
NOT
AND       M04101	// 10_R_P&P Y PICK 2nd
AND       P0005E	// R_P&P DOWN
AND       P00160	// R_P&P 1st EJECT ON
AND       P00140	// R_1st DIE VACUUM EJECTOR ON
LOADP     T0054	// RT_AUTO RUN 0.6
AND NOT   M06611	// R_1st DIE VACUUM CHECK ON
AND NOT   M1261A	// R_1st DIE VC CLEAR OFF
OR LOAD
OUT       M12622	// R_1st MAND VC OFF

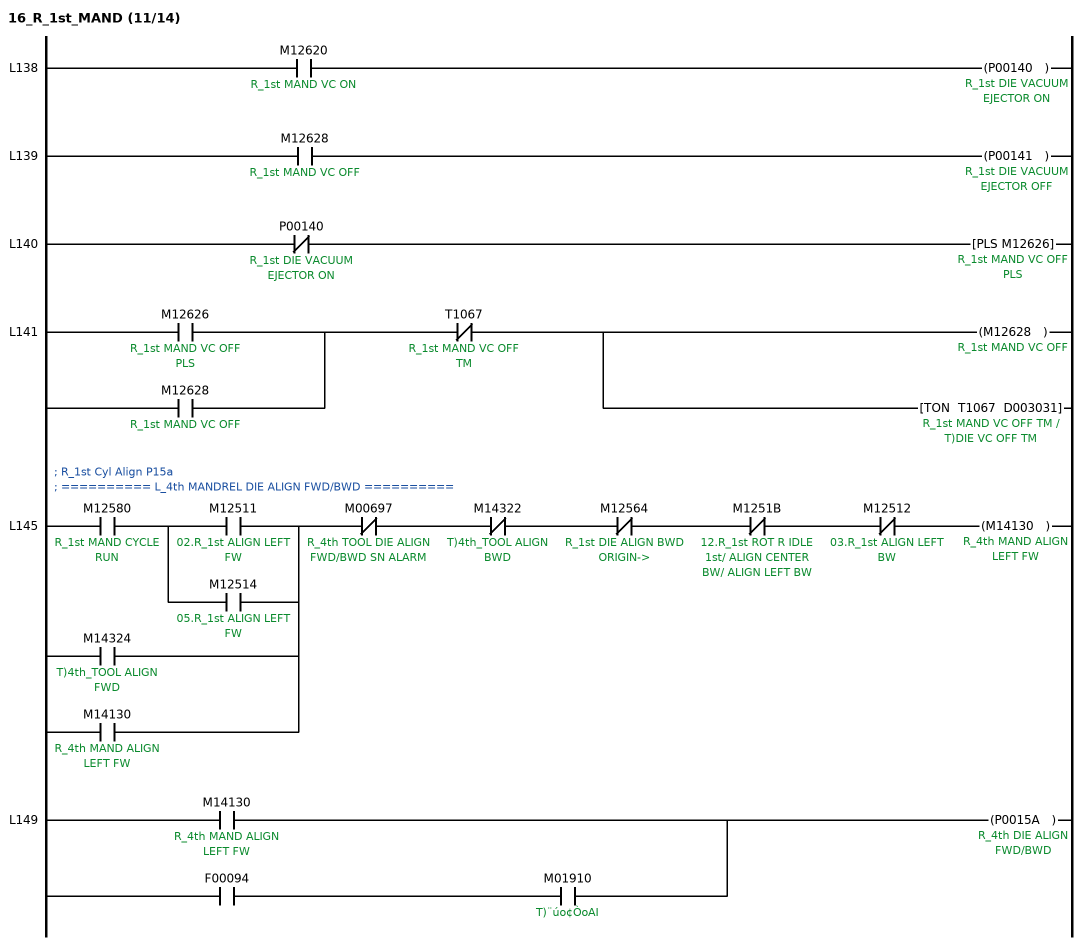
; L138
LOAD      M12620	// R_1st MAND VC ON
OUT       P00140	// R_1st DIE VACUUM EJECTOR ON
; L139
LOAD      M12628	// R_1st MAND VC OFF
OUT       P00141	// R_1st DIE VACUUM EJECTOR OFF
; L140
LOAD NOT  P00140	// R_1st DIE VACUUM EJECTOR ON
OUTP      M12626	// R_1st MAND VC OFF PLS
; L141
LOAD      M12626	// R_1st MAND VC OFF PLS
OR        M12628	// R_1st MAND VC OFF
AND NOT   T1067	// R_1st MAND VC OFF TM
OUT       M12628	// R_1st MAND VC OFF
TON       T1067 D003031	// R_1st MAND VC OFF TM / T)DIE VC OFF TM
// R_1st Cyl Align P15a
// ========== L_4th MANDREL DIE ALIGN FWD/BWD ==========
; L145
LOAD      M12580	// R_1st MAND CYCLE RUN
LOAD      M12511	// 02.R_1st ALIGN LEFT FW
OR        M12514	// 05.R_1st ALIGN LEFT FW
AND LOAD
OR        M14324	// T)4th_TOOL ALIGN FWD
OR        M14130	// R_4th MAND ALIGN LEFT FW
AND NOT   M00697	// R_4th TOOL DIE ALIGN FWD/BWD SN ALARM
AND NOT   M14322	// T)4th_TOOL ALIGN BWD
AND NOT   M12564	// R_1st DIE ALIGN BWD ORIGIN->
AND NOT   M1251B	// 12.R_1st ROT R IDLE 1st/ ALIGN CENTER BW/ ALIGN LEFT BW
AND NOT   M12512	// 03.R_1st ALIGN LEFT BW
OUT       M14130	// R_4th MAND ALIGN LEFT FW
; L149
LOAD      M14130	// R_4th MAND ALIGN LEFT FW
LOAD      F00094
AND       M01910	// T)¨úo¢ÒoAI
OR LOAD
OUT       P0015A	// R_4th DIE ALIGN FWD/BWD

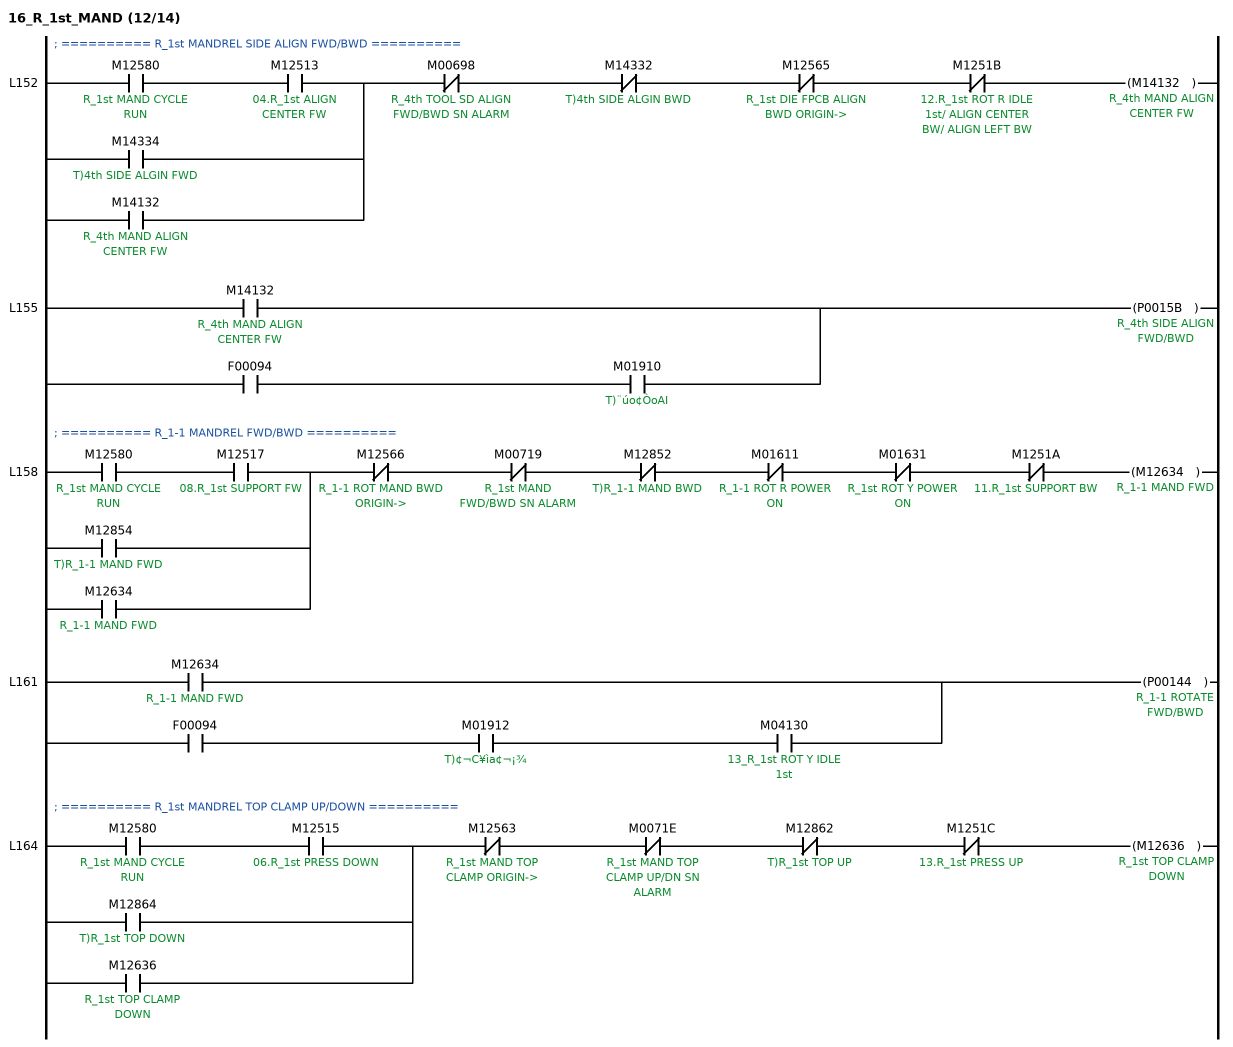
// ========== R_1st MANDREL SIDE ALIGN FWD/BWD ==========
; L152
LOAD      M12580	// R_1st MAND CYCLE RUN
AND       M12513	// 04.R_1st ALIGN CENTER FW
OR        M14334	// T)4th SIDE ALGIN FWD
OR        M14132	// R_4th MAND ALIGN CENTER FW
AND NOT   M00698	// R_4th TOOL SD ALIGN FWD/BWD SN ALARM
AND NOT   M14332	// T)4th SIDE ALGIN BWD
AND NOT   M12565	// R_1st DIE FPCB ALIGN BWD ORIGIN->
AND NOT   M1251B	// 12.R_1st ROT R IDLE 1st/ ALIGN CENTER BW/ ALIGN LEFT BW
OUT       M14132	// R_4th MAND ALIGN CENTER FW
; L155
LOAD      M14132	// R_4th MAND ALIGN CENTER FW
LOAD      F00094
AND       M01910	// T)¨úo¢ÒoAI
OR LOAD
OUT       P0015B	// R_4th SIDE ALIGN FWD/BWD
// ========== R_1-1 MANDREL FWD/BWD ==========
; L158
LOAD      M12580	// R_1st MAND CYCLE RUN
AND       M12517	// 08.R_1st SUPPORT FW
OR        M12854	// T)R_1-1 MAND FWD
OR        M12634	// R_1-1 MAND FWD
AND NOT   M12566	// R_1-1 ROT MAND BWD ORIGIN->
AND NOT   M00719	// R_1st MAND FWD/BWD SN ALARM
AND NOT   M12852	// T)R_1-1 MAND BWD
AND NOT   M01611	// R_1-1 ROT R POWER ON
AND NOT   M01631	// R_1st ROT Y POWER ON
AND NOT   M1251A	// 11.R_1st SUPPORT BW
OUT       M12634	// R_1-1 MAND FWD
; L161
LOAD      M12634	// R_1-1 MAND FWD
LOAD      F00094
AND       M01912	// T)¢¬C¥ìa¢¬¡¾
AND       M04130	// 13_R_1st ROT Y IDLE 1st
OR LOAD
OUT       P00144	// R_1-1 ROTATE FWD/BWD
// ========== R_1st MANDREL TOP CLAMP UP/DOWN ==========
; L164
LOAD      M12580	// R_1st MAND CYCLE RUN
AND       M12515	// 06.R_1st PRESS DOWN
OR        M12864	// T)R_1st TOP DOWN
OR        M12636	// R_1st TOP CLAMP DOWN
AND NOT   M12563	// R_1st MAND TOP CLAMP ORIGIN->
AND NOT   M0071E	// R_1st MAND TOP CLAMP UP/DN SN ALARM
AND NOT   M12862	// T)R_1st TOP UP
AND NOT   M1251C	// 13.R_1st PRESS UP
OUT       M12636	// R_1st TOP CLAMP DOWN

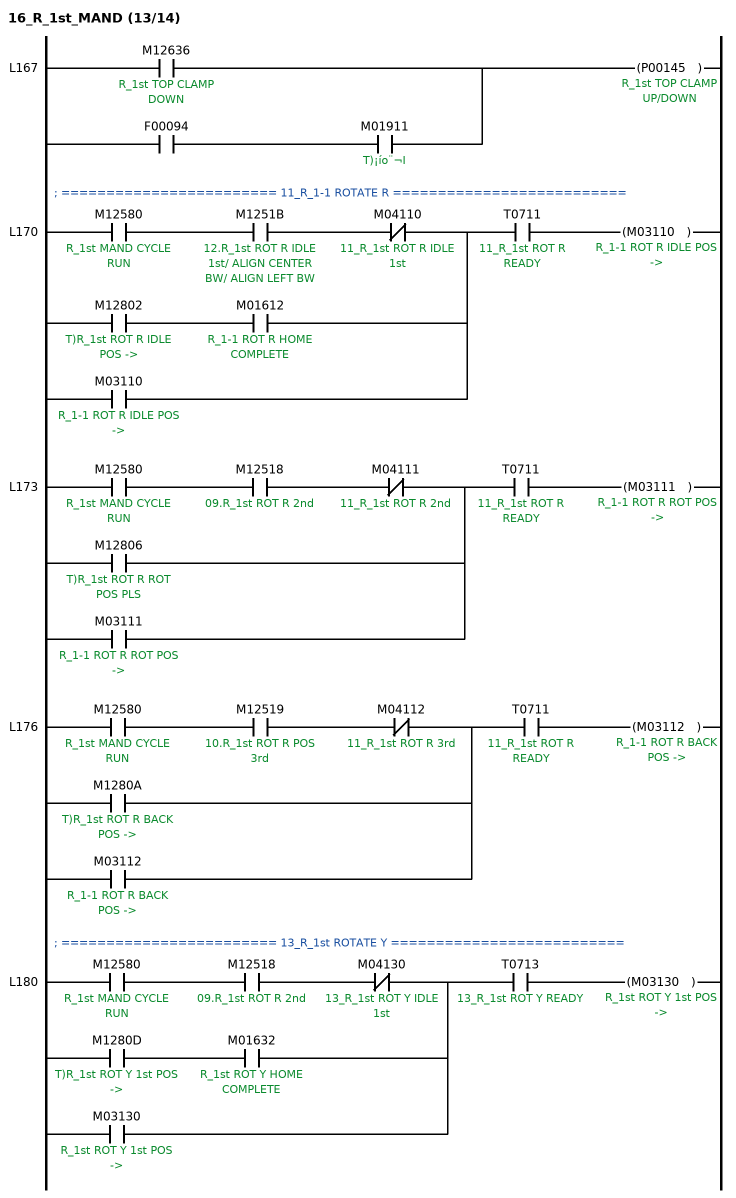
; L167
LOAD      M12636	// R_1st TOP CLAMP DOWN
LOAD      F00094
AND       M01911	// T)¡ío¨¬I
OR LOAD
OUT       P00145	// R_1st TOP CLAMP UP/DOWN
// ======================== 11_R_1-1 ROTATE R ==========================
; L170
LOAD      M12580	// R_1st MAND CYCLE RUN
AND       M1251B	// 12.R_1st ROT R IDLE 1st/ ALIGN CENTER BW/ ALIGN LEFT BW
AND NOT   M04110	// 11_R_1st ROT R IDLE 1st
LOAD      M12802	// T)R_1st ROT R IDLE POS ->
AND       M01612	// R_1-1 ROT R HOME COMPLETE
OR LOAD
OR        M03110	// R_1-1 ROT R IDLE POS ->
AND       T0711	// 11_R_1st ROT R READY
OUT       M03110	// R_1-1 ROT R IDLE POS ->
; L173
LOAD      M12580	// R_1st MAND CYCLE RUN
AND       M12518	// 09.R_1st ROT R 2nd
AND NOT   M04111	// 11_R_1st ROT R 2nd
OR        M12806	// T)R_1st ROT R ROT POS PLS
OR        M03111	// R_1-1 ROT R ROT POS ->
AND       T0711	// 11_R_1st ROT R READY
OUT       M03111	// R_1-1 ROT R ROT POS ->
; L176
LOAD      M12580	// R_1st MAND CYCLE RUN
AND       M12519	// 10.R_1st ROT R POS 3rd
AND NOT   M04112	// 11_R_1st ROT R 3rd
OR        M1280A	// T)R_1st ROT R BACK POS ->
OR        M03112	// R_1-1 ROT R BACK POS ->
AND       T0711	// 11_R_1st ROT R READY
OUT       M03112	// R_1-1 ROT R BACK POS ->
// ======================== 13_R_1st ROTATE Y ==========================
; L180
LOAD      M12580	// R_1st MAND CYCLE RUN
AND       M12518	// 09.R_1st ROT R 2nd
AND NOT   M04130	// 13_R_1st ROT Y IDLE 1st
LOAD      M1280D	// T)R_1st ROT Y 1st POS ->
AND       M01632	// R_1st ROT Y HOME COMPLETE
OR LOAD
OR        M03130	// R_1st ROT Y 1st POS ->
AND       T0713	// 13_R_1st ROT Y READY
OUT       M03130	// R_1st ROT Y 1st POS ->

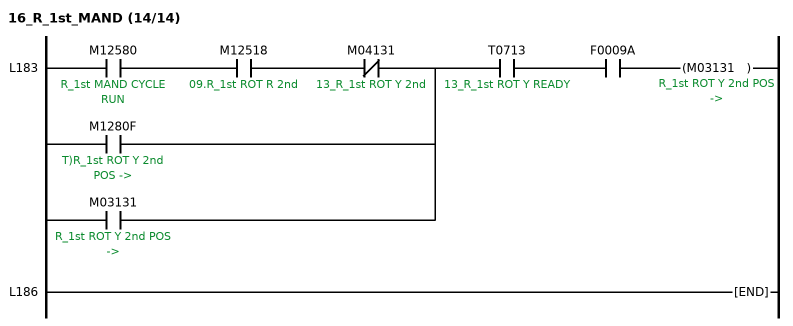
; L183
LOAD      M12580	// R_1st MAND CYCLE RUN
AND       M12518	// 09.R_1st ROT R 2nd
AND NOT   M04131	// 13_R_1st ROT Y 2nd
OR        M1280F	// T)R_1st ROT Y 2nd POS ->
OR        M03131	// R_1st ROT Y 2nd POS ->
AND       T0713	// 13_R_1st ROT Y READY
AND       F0009A
OUT       M03131	// R_1st ROT Y 2nd POS ->
; L186
END

PROGRAM 17_R_2nd_MAND (task: ¨ö¨¬A¥ì CA¡¤I¡¾¡¿¡¤¡Í)

